RoboDK station: Config_3.rdk

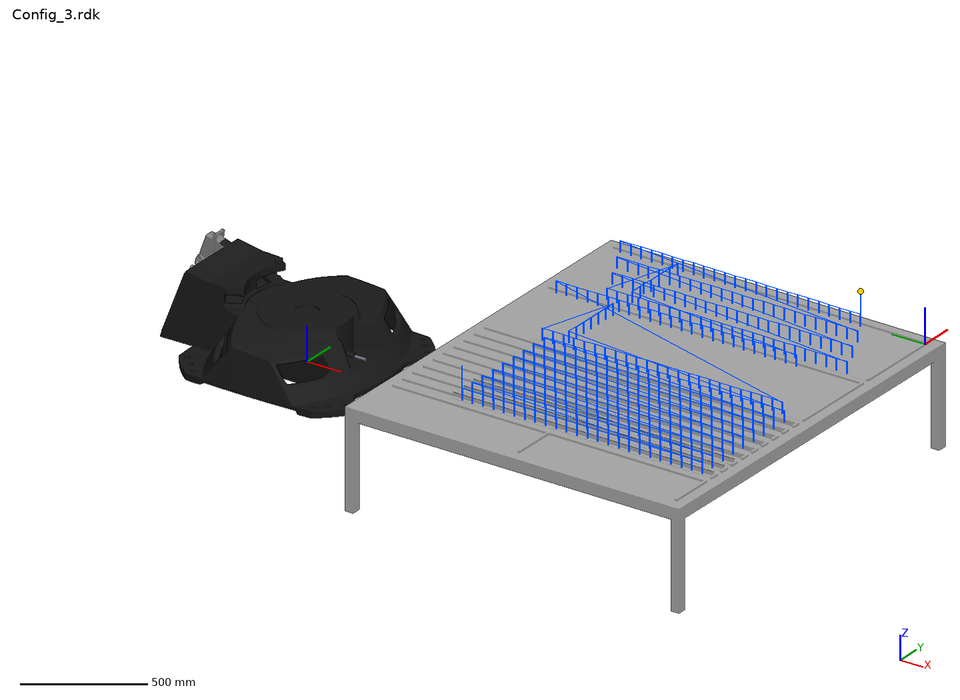
[picture v0: the station drawn from its stored meshes, robots at their saved joint values, targets as dots, program paths as lines]
Station Config_3 (saved by RoboDK 5.2.3). Poses are relative to the parent item; angles as X-Y-Z fixed-axis rotations.
  - frame KUKA KR 210 R2700 extra Base at (0, 0, 0) mm
    - robot KUKA KR 210 R2700 extra: 6 axes, payload 210 kg, reach 2696 mm, repeatability 0.06 mm, weight 1068 kg
        joint limits [-185, -140, -120, -350, -125, -350] to [185, -5, 155, 350, 125, 350]; home [0, -90, 90, 0, 0, 0]; saved at [38.533, -84.893, 130.139, 228.276, 56.581, -211.701]
      - tool Spindle, TCP at (278.6, 0, 88) mm, rotated rx 0 ry 90 rz 0 deg, size 85 x 346.5 x 128 mm
  - frame Corner First Plate at (2495, 660, 510.8) mm, rotated rx 0 ry 0 rz 90 deg
  - object Table 3 at (1700, -800, 455) mm, rotated rx 0 ry 0 rz 90 deg, size 1820 x 1600 x 475 mm, geometry from Table 3.stl
  - object Config_3 at (2495, 660, 510.8) mm, rotated rx 0 ry 0 rz 90 deg
  - machining project Path1 settings: rotZ(0) | rotX(0)*rotY(0) | rotz(0) | onStart | onPathStart | onApproach | onPoint | onRetract | onFinish | SetRPM(%1) | SetTool(%1) | Extruder(%1) | default | default | OutOnMov(%1) | OutOffMov(%1) | onPathFinish | M_RunCode(%1)
  - program Path1 (1131 instructions, listed below)
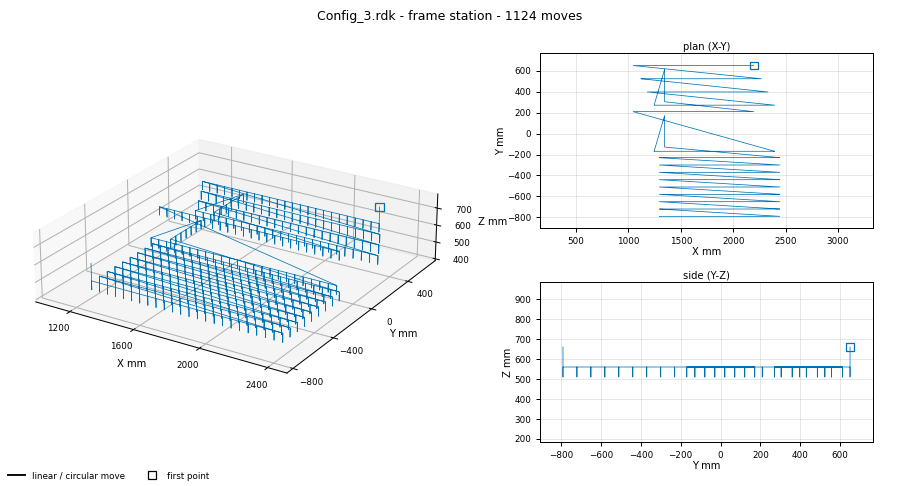
[picture p0: tool path of Config_3.rdk in frame station, 1124 of 1124 moves have a stored position in this frame; points joined in program order, loops and branches not executed]

--- program Path1 (robot KUKA KR 210 R2700 extra) ---
  Smooth(1)
  Set speed (1000.0 mm/s)
  Set Ref.: Corner First Plate
  Set Tool: Spindle
  Show Spindle
  MoveJ 1 to (-10.8, 300, 150) mm, rotated rx 180 ry 0 rz 90 deg; joints [-18.939, -55.022, 87.438, 147.377, 37.015, -152.928]
  MoveL 2 to (-10.8, 300, 150) mm, rotated rx 180 ry 0 rz 90 deg; joints [-18.939, -55.022, 87.438, 147.377, 37.015, -152.928]
  MoveL 3 to (-10.8, 300, 50) mm, rotated rx -180 ry 0 rz 90 deg; joints [-18.939, -52.073, 88.328, 149.877, 40.293, -156.128]
  MoveL 4 to (-10.8, 300, 50) mm, rotated rx -180 ry 0 rz 90 deg; joints [-18.939, -52.073, 88.328, 149.877, 40.293, -156.128]
  Set speed (150.0 mm/s)
  MoveL 5 to (-10.8, 300, -0.5) mm, rotated rx 180 ry 0 rz 90 deg; joints [-18.939, -50.484, 88.62, 150.941, 41.929, -157.54]
  MoveL 6 to (-10.8, 300, 50) mm, rotated rx -180 ry 0 rz 90 deg; joints [-18.939, -52.073, 88.328, 149.877, 40.293, -156.128]
  MoveL 7 to (-10.8, 350, 50) mm, rotated rx 180 ry 0 rz 90 deg; joints [-19.415, -53.906, 91.518, 149.994, 41.659, -156.663]
  MoveL 8 to (-10.8, 350, -0.5) mm, rotated rx 180 ry 0 rz 90 deg; joints [-19.415, -52.267, 91.81, 151.032, 43.339, -158.069]
  MoveL 9 to (-10.8, 350, 50) mm, rotated rx 180 ry 0 rz 90 deg; joints [-19.415, -53.906, 91.518, 149.994, 41.659, -156.663]
  MoveL 10 to (-10.8, 400, 50) mm, rotated rx 180 ry 0 rz 90 deg; joints [-19.914, -55.704, 94.616, 150.026, 42.981, -157.123]
  MoveL 11 to (-10.8, 400, -0.5) mm, rotated rx -180 ry 0 rz 90 deg; joints [-19.914, -54.013, 94.91, 151.042, 44.709, -158.532]
  MoveL 12 to (-10.8, 400, 50) mm, rotated rx 180 ry 0 rz 90 deg; joints [-19.914, -55.704, 94.616, 150.026, 42.981, -157.123]
  MoveL 13 to (-10.8, 450, 50) mm, rotated rx 180 ry 0 rz 90 deg; joints [-20.439, -57.473, 97.631, 149.977, 44.262, -157.517]
  MoveL 14 to (-10.8, 450, -0.5) mm, rotated rx 180 ry 0 rz 90 deg; joints [-20.439, -55.727, 97.926, 150.978, 46.038, -158.936]
  MoveL 15 to (-10.8, 450, 50) mm, rotated rx 180 ry 0 rz 90 deg; joints [-20.439, -57.473, 97.631, 149.977, 44.262, -157.517]
  MoveL 16 to (-10.8, 500, 50) mm, rotated rx -180 ry 0 rz 90 deg; joints [-20.991, -59.217, 100.569, 149.854, 45.504, -157.852]
  MoveL 17 to (-10.8, 500, -0.5) mm, rotated rx 180 ry 0 rz 90 deg; joints [-20.991, -57.414, 100.867, 150.844, 47.331, -159.288]
  MoveL 18 to (-10.8, 500, 50) mm, rotated rx -180 ry 0 rz 90 deg; joints [-20.991, -59.217, 100.569, 149.854, 45.504, -157.852]
  MoveL 19 to (-10.8, 550, 50) mm, rotated rx 180 ry 0 rz 90 deg; joints [-21.572, -60.942, 103.435, 149.66, 46.709, -158.133]
  MoveL 20 to (-10.8, 550, -0.5) mm, rotated rx 180 ry 0 rz 90 deg; joints [-21.572, -59.078, 103.738, 150.643, 48.588, -159.592]
  MoveL 21 to (-10.8, 550, 50) mm, rotated rx 180 ry 0 rz 90 deg; joints [-21.572, -60.942, 103.435, 149.66, 46.709, -158.133]
  MoveL 22 to (-10.8, 600, 50) mm, rotated rx 180 ry 0 rz 90 deg; joints [-22.185, -62.649, 106.236, 149.397, 47.878, -158.362]
  MoveL 23 to (-10.8, 600, -0.5) mm, rotated rx 180 ry 0 rz 90 deg; joints [-22.185, -60.721, 106.543, 150.377, 49.812, -159.851]
  MoveL 24 to (-10.8, 600, 50) mm, rotated rx 180 ry 0 rz 90 deg; joints [-22.185, -62.649, 106.236, 149.397, 47.878, -158.362]
  MoveL 25 to (-10.8, 650, 50) mm, rotated rx 180 ry 0 rz 90 deg; joints [-22.832, -64.344, 108.975, 149.067, 49.013, -158.542]
  MoveL 26 to (-10.8, 650, -0.5) mm, rotated rx 180 ry 0 rz 90 deg; joints [-22.832, -62.348, 109.287, 150.048, 51.003, -160.069]
  MoveL 27 to (-10.8, 650, 50) mm, rotated rx 180 ry 0 rz 90 deg; joints [-22.832, -64.344, 108.975, 149.067, 49.013, -158.542]
  MoveL 28 to (-10.8, 700, 50) mm, rotated rx -180 ry 0 rz 90 deg; joints [-23.515, -66.029, 111.655, 148.669, 50.113, -158.676]
  MoveL 29 to (-10.8, 700, -0.5) mm, rotated rx 180 ry 0 rz 90 deg; joints [-23.515, -63.961, 111.973, 149.655, 52.163, -160.247]
  MoveL 30 to (-10.8, 700, 50) mm, rotated rx -180 ry 0 rz 90 deg; joints [-23.515, -66.029, 111.655, 148.669, 50.113, -158.676]
  MoveL 31 to (-10.8, 750, 50) mm, rotated rx 180 ry 0 rz 90 deg; joints [-24.238, -67.708, 114.279, 148.204, 51.181, -158.763]
  MoveL 32 to (-10.8, 750, -0.5) mm, rotated rx 180 ry 0 rz 90 deg; joints [-24.238, -65.564, 114.604, 149.198, 53.292, -160.386]
  MoveL 33 to (-10.8, 750, 50) mm, rotated rx 180 ry 0 rz 90 deg; joints [-24.238, -67.708, 114.279, 148.204, 51.181, -158.763]
  MoveL 34 to (-10.8, 800, 50) mm, rotated rx -180 ry 0 rz 90 deg; joints [-25.003, -69.384, 116.85, 147.669, 52.216, -158.805]
  MoveL 35 to (-10.8, 800, -0.5) mm, rotated rx 180 ry 0 rz 90 deg; joints [-25.003, -67.159, 117.183, 148.675, 54.391, -160.488]
  MoveL 36 to (-10.8, 800, 50) mm, rotated rx -180 ry 0 rz 90 deg; joints [-25.003, -69.384, 116.85, 147.669, 52.216, -158.805]
  MoveL 37 to (-10.8, 850, 50) mm, rotated rx -180 ry 0 rz 90 deg; joints [-25.816, -71.061, 119.369, 147.064, 53.22, -158.799]
  MoveL 38 to (-10.8, 850, -0.5) mm, rotated rx 180 ry 0 rz 90 deg; joints [-25.816, -68.749, 119.711, 148.085, 55.46, -160.551]
  MoveL 39 to (-10.8, 850, 50) mm, rotated rx -180 ry 0 rz 90 deg; joints [-25.816, -71.061, 119.369, 147.064, 53.22, -158.799]
  MoveL 40 to (-10.8, 900, 50) mm, rotated rx 180 ry 0 rz 90 deg; joints [-26.678, -72.742, 121.838, 146.383, 54.192, -158.746]
  MoveL 41 to (-10.8, 900, -0.5) mm, rotated rx -180 ry 0 rz 90 deg; joints [-26.678, -70.337, 122.19, 147.424, 56.501, -160.575]
  MoveL 42 to (-10.8, 900, 50) mm, rotated rx 180 ry 0 rz 90 deg; joints [-26.678, -72.742, 121.838, 146.383, 54.192, -158.746]
  MoveL 43 to (-10.8, 950, 50) mm, rotated rx -180 ry 0 rz 90 deg; joints [-27.596, -74.43, 124.259, 145.626, 55.132, -158.641]
  MoveL 44 to (-10.8, 950, -0.5) mm, rotated rx -180 ry 0 rz 90 deg; joints [-27.596, -71.926, 124.621, 146.689, 57.513, -160.559]
  MoveL 45 to (-10.8, 950, 50) mm, rotated rx -180 ry 0 rz 90 deg; joints [-27.596, -74.43, 124.259, 145.626, 55.132, -158.641]
  MoveL 46 to (-10.8, 1000, 50) mm, rotated rx 180 ry 0 rz 90 deg; joints [-28.574, -76.128, 126.631, 144.786, 56.043, -158.484]
  MoveL 47 to (-10.8, 1000, -0.5) mm, rotated rx 180 ry 0 rz 90 deg; joints [-28.574, -73.519, 127.005, 145.877, 58.497, -160.501]
  MoveL 48 to (-10.8, 1000, 50) mm, rotated rx 180 ry 0 rz 90 deg; joints [-28.574, -76.128, 126.631, 144.786, 56.043, -158.484]
  MoveL 49 to (-10.8, 1050, 50) mm, rotated rx -180 ry 0 rz 90 deg; joints [-29.617, -77.842, 128.955, 143.858, 56.923, -158.269]
  MoveL 50 to (-10.8, 1050, -0.5) mm, rotated rx 180 ry 0 rz 90 deg; joints [-29.617, -75.119, 129.342, 144.981, 59.453, -160.398]
  MoveL 51 to (-10.8, 1050, 50) mm, rotated rx -180 ry 0 rz 90 deg; joints [-29.617, -77.842, 128.955, 143.858, 56.923, -158.269]
  MoveL 52 to (-10.8, 1100, 50) mm, rotated rx 180 ry 0 rz 90 deg; joints [-30.732, -79.573, 131.231, 142.838, 57.775, -157.992]
  MoveL 53 to (-10.8, 1100, -0.5) mm, rotated rx -180 ry 0 rz 90 deg; joints [-30.732, -76.729, 131.632, 143.997, 60.382, -160.246]
  MoveL 54 to (-10.8, 1100, 50) mm, rotated rx 180 ry 0 rz 90 deg; joints [-30.732, -79.573, 131.231, 142.838, 57.775, -157.992]
  MoveL 55 to (-10.8, 1150, 50) mm, rotated rx 180 ry 0 rz 90 deg; joints [-31.924, -81.327, 133.457, 141.718, 58.599, -157.647]
  MoveL 56 to (-10.8, 1150, -0.5) mm, rotated rx 180 ry 0 rz 90 deg; joints [-31.924, -78.352, 133.874, 142.918, 61.284, -160.042]
  MoveL 57 to (-10.8, 1150, 50) mm, rotated rx 180 ry 0 rz 90 deg; joints [-31.924, -81.327, 133.457, 141.718, 58.599, -157.647]
  MoveL 58 to (-10.8, 1200, 50) mm, rotated rx 180 ry 0 rz 90 deg; joints [-33.202, -83.108, 135.634, 140.49, 59.397, -157.227]
  MoveL 59 to (-10.8, 1200, -0.5) mm, rotated rx 180 ry 0 rz 90 deg; joints [-33.202, -79.993, 136.068, 141.737, 62.161, -159.78]
  MoveL 60 to (-10.8, 1200, 50) mm, rotated rx 180 ry 0 rz 90 deg; joints [-33.202, -83.108, 135.634, 140.49, 59.397, -157.227]
  MoveL 61 to (-10.8, 1250, 50) mm, rotated rx -180 ry 0 rz 90 deg; joints [-34.574, -84.92, 137.758, 139.147, 60.172, -156.726]
  MoveL 62 to (-10.8, 1250, -0.5) mm, rotated rx -180 ry 0 rz 90 deg; joints [-34.574, -81.654, 138.211, 140.446, 63.014, -159.455]
  MoveL 63 to (-10.8, 1250, 50) mm, rotated rx -180 ry 0 rz 90 deg; joints [-34.574, -84.92, 137.758, 139.147, 60.172, -156.726]
  MoveL 64 to (-10.8, 1300, 50) mm, rotated rx 180 ry 0 rz 90 deg; joints [-36.047, -86.767, 139.828, 137.68, 60.929, -156.133]
  MoveL 65 to (-10.8, 1300, -0.5) mm, rotated rx 180 ry 0 rz 90 deg; joints [-36.047, -83.339, 140.302, 139.037, 63.846, -159.059]
  MoveL 66 to (-10.8, 1300, 50) mm, rotated rx 180 ry 0 rz 90 deg; joints [-36.047, -86.767, 139.828, 137.68, 60.929, -156.133]
  MoveL 67 to (-10.8, 1350, 50) mm, rotated rx 180 ry 0 rz 90 deg; joints [-37.633, -88.655, 141.842, 136.078, 61.671, -155.439]
  MoveL 68 to (-10.8, 1350, -0.5) mm, rotated rx 180 ry 0 rz 90 deg; joints [-37.633, -85.052, 142.339, 137.499, 64.659, -158.585]
  MoveL 69 to (-10.8, 1350, 50) mm, rotated rx 180 ry 0 rz 90 deg; joints [-37.633, -88.655, 141.842, 136.078, 61.671, -155.439]
  MoveL 70 to (-10.8, 1400, 50) mm, rotated rx -180 ry 0 rz 90 deg; joints [-39.341, -90.587, 143.795, 134.333, 62.407, -154.634]
  MoveL 71 to (-10.8, 1400, -0.5) mm, rotated rx 180 ry 0 rz 90 deg; joints [-39.341, -86.798, 144.317, 135.822, 65.461, -158.023]
  MoveL 72 to (-10.8, 1400, 50) mm, rotated rx -180 ry 0 rz 90 deg; joints [-39.341, -90.587, 143.795, 134.333, 62.407, -154.634]
  MoveL 73 to (-10.8, 1450, 50) mm, rotated rx 180 ry 0 rz 90 deg; joints [-41.184, -92.567, 145.684, 132.434, 63.147, -153.707]
  MoveL 74 to (-10.8, 1450, -0.5) mm, rotated rx -180 ry 0 rz 90 deg; joints [-41.184, -88.578, 146.233, 133.998, 66.256, -157.364]
  MoveL 75 to (-10.8, 1450, 50) mm, rotated rx 180 ry 0 rz 90 deg; joints [-41.184, -92.567, 145.684, 132.434, 63.147, -153.707]
  MoveL 76 to (-136.94, 226.53, 50) mm, rotated rx -180 ry 0 rz 90 deg; joints [-14.902, -50.749, 86.003, 155.248, 37.896, -160.007]
  MoveL 77 to (-136.94, 226.53, -0.5) mm, rotated rx 180 ry 0 rz 90 deg; joints [-14.902, -49.194, 86.295, 156.194, 39.579, -161.22]
  MoveL 78 to (-136.94, 226.53, 50) mm, rotated rx -180 ry 0 rz 90 deg; joints [-14.902, -50.749, 86.003, 155.248, 37.896, -160.007]
  MoveL 79 to (-136.94, 276.53, 50) mm, rotated rx -180 ry 0 rz 90 deg; joints [-15.273, -52.646, 89.329, 155.434, 39.319, -160.525]
  MoveL 80 to (-136.94, 276.53, -0.5) mm, rotated rx 180 ry 0 rz 90 deg; joints [-15.273, -51.042, 89.62, 156.351, 41.049, -161.724]
  MoveL 81 to (-136.94, 276.53, 50) mm, rotated rx -180 ry 0 rz 90 deg; joints [-15.273, -52.646, 89.329, 155.434, 39.319, -160.525]
  MoveL 82 to (-136.94, 326.53, 50) mm, rotated rx -180 ry 0 rz 90 deg; joints [-15.663, -54.506, 92.556, 155.538, 40.691, -160.969]
  MoveL 83 to (-136.94, 326.53, -0.5) mm, rotated rx -180 ry 0 rz 90 deg; joints [-15.663, -52.85, 92.848, 156.432, 42.471, -162.163]
  MoveL 84 to (-136.94, 326.53, 50) mm, rotated rx -180 ry 0 rz 90 deg; joints [-15.663, -54.506, 92.556, 155.538, 40.691, -160.969]
  MoveL 85 to (-136.94, 376.53, 50) mm, rotated rx 180 ry 0 rz 90 deg; joints [-16.072, -56.334, 95.694, 155.568, 42.016, -161.349]
  MoveL 86 to (-136.94, 376.53, -0.5) mm, rotated rx -180 ry 0 rz 90 deg; joints [-16.072, -54.624, 95.988, 156.444, 43.847, -162.545]
  MoveL 87 to (-136.94, 376.53, 50) mm, rotated rx 180 ry 0 rz 90 deg; joints [-16.072, -56.334, 95.694, 155.568, 42.016, -161.349]
  MoveL 88 to (-136.94, 426.53, 50) mm, rotated rx 180 ry 0 rz 90 deg; joints [-16.503, -58.136, 98.751, 155.529, 43.296, -161.673]
  MoveL 89 to (-136.94, 426.53, -0.5) mm, rotated rx -180 ry 0 rz 90 deg; joints [-16.503, -56.369, 99.048, 156.392, 45.18, -162.878]
  MoveL 90 to (-136.94, 426.53, 50) mm, rotated rx 180 ry 0 rz 90 deg; joints [-16.503, -58.136, 98.751, 155.529, 43.296, -161.673]
  MoveL 91 to (-136.94, 476.53, 50) mm, rotated rx 180 ry 0 rz 90 deg; joints [-16.957, -59.916, 101.734, 155.426, 44.532, -161.945]
  MoveL 92 to (-136.94, 476.53, -0.5) mm, rotated rx -180 ry 0 rz 90 deg; joints [-16.957, -58.088, 102.034, 156.281, 46.473, -163.165]
  MoveL 93 to (-136.94, 476.53, 50) mm, rotated rx 180 ry 0 rz 90 deg; joints [-16.957, -59.916, 101.734, 155.426, 44.532, -161.945]
  MoveL 94 to (-136.94, 526.53, 50) mm, rotated rx 180 ry 0 rz 90 deg; joints [-17.435, -61.679, 104.649, 155.262, 45.726, -162.17]
  MoveL 95 to (-136.94, 526.53, -0.5) mm, rotated rx 180 ry 0 rz 90 deg; joints [-17.435, -59.788, 104.954, 156.113, 47.727, -163.411]
  MoveL 96 to (-136.94, 526.53, 50) mm, rotated rx 180 ry 0 rz 90 deg; joints [-17.435, -61.679, 104.649, 155.262, 45.726, -162.17]
  MoveL 97 to (-136.94, 576.53, 50) mm, rotated rx -180 ry 0 rz 90 deg; joints [-17.941, -63.429, 107.501, 155.038, 46.88, -162.35]
  MoveL 98 to (-136.94, 576.53, -0.5) mm, rotated rx -180 ry 0 rz 90 deg; joints [-17.941, -61.47, 107.811, 155.889, 48.944, -163.619]
  MoveL 99 to (-136.94, 576.53, 50) mm, rotated rx -180 ry 0 rz 90 deg; joints [-17.941, -63.429, 107.501, 155.038, 46.88, -162.35]
  MoveL 100 to (-136.94, 626.53, 50) mm, rotated rx -180 ry 0 rz 90 deg; joints [-18.476, -65.17, 110.295, 154.756, 47.994, -162.488]
  MoveL 101 to (-136.94, 626.53, -0.5) mm, rotated rx -180 ry 0 rz 90 deg; joints [-18.476, -63.14, 110.61, 155.61, 50.124, -163.791]
  MoveL 102 to (-136.94, 626.53, 50) mm, rotated rx -180 ry 0 rz 90 deg; joints [-18.476, -65.17, 110.295, 154.756, 47.994, -162.488]
  MoveL 103 to (-136.94, 676.53, 50) mm, rotated rx -180 ry 0 rz 90 deg; joints [-19.042, -66.907, 113.033, 154.415, 49.069, -162.584]
  MoveL 104 to (-136.94, 676.53, -0.5) mm, rotated rx 180 ry 0 rz 90 deg; joints [-19.042, -64.8, 113.355, 155.276, 51.268, -163.929]
  MoveL 105 to (-136.94, 676.53, 50) mm, rotated rx -180 ry 0 rz 90 deg; joints [-19.042, -66.907, 113.033, 154.415, 49.069, -162.584]
  MoveL 106 to (-136.94, 726.53, 50) mm, rotated rx 180 ry 0 rz 90 deg; joints [-19.643, -68.643, 115.719, 154.014, 50.104, -162.639]
  MoveL 107 to (-136.94, 726.53, -0.5) mm, rotated rx -180 ry 0 rz 90 deg; joints [-19.643, -66.454, 116.049, 154.886, 52.376, -164.032]
  MoveL 108 to (-136.94, 726.53, 50) mm, rotated rx 180 ry 0 rz 90 deg; joints [-19.643, -68.643, 115.719, 154.014, 50.104, -162.639]
  MoveL 109 to (-136.94, 776.53, 50) mm, rotated rx 180 ry 0 rz 90 deg; joints [-20.281, -70.382, 118.355, 153.551, 51.099, -162.652]
  MoveL 110 to (-136.94, 776.53, -0.5) mm, rotated rx -180 ry 0 rz 90 deg; joints [-20.281, -68.106, 118.694, 154.439, 53.45, -164.101]
  MoveL 111 to (-136.94, 776.53, 50) mm, rotated rx 180 ry 0 rz 90 deg; joints [-20.281, -70.382, 118.355, 153.551, 51.099, -162.652]
  MoveL 112 to (-136.94, 826.53, 50) mm, rotated rx 180 ry 0 rz 90 deg; joints [-20.96, -72.129, 120.945, 153.024, 52.055, -162.621]
  MoveL 113 to (-136.94, 826.53, -0.5) mm, rotated rx 180 ry 0 rz 90 deg; joints [-20.96, -69.759, 121.293, 153.93, 54.487, -164.135]
  MoveL 114 to (-136.94, 826.53, 50) mm, rotated rx 180 ry 0 rz 90 deg; joints [-20.96, -72.129, 120.945, 153.024, 52.055, -162.621]
  MoveL 115 to (-136.94, 876.53, 50) mm, rotated rx -180 ry 0 rz 90 deg; joints [-21.684, -73.888, 123.489, 152.43, 52.969, -162.544]
  MoveL 116 to (-136.94, 876.53, -0.5) mm, rotated rx -180 ry 0 rz 90 deg; joints [-21.684, -71.417, 123.848, 153.359, 55.489, -164.134]
  MoveL 117 to (-136.94, 876.53, 50) mm, rotated rx -180 ry 0 rz 90 deg; joints [-21.684, -73.888, 123.489, 152.43, 52.969, -162.544]
  MoveL 118 to (-136.94, 926.53, 50) mm, rotated rx -180 ry 0 rz 90 deg; joints [-22.457, -75.664, 125.989, 151.763, 53.842, -162.419]
  MoveL 119 to (-136.94, 926.53, -0.5) mm, rotated rx 180 ry 0 rz 90 deg; joints [-22.457, -73.084, 126.36, 152.721, 56.453, -164.094]
  MoveL 120 to (-136.94, 926.53, 50) mm, rotated rx -180 ry 0 rz 90 deg; joints [-22.457, -75.664, 125.989, 151.763, 53.842, -162.419]
  MoveL 121 to (-136.94, 976.53, 50) mm, rotated rx -180 ry 0 rz 90 deg; joints [-23.284, -77.462, 128.446, 151.02, 54.671, -162.241]
  MoveL 122 to (-136.94, 976.53, -0.5) mm, rotated rx 180 ry 0 rz 90 deg; joints [-23.284, -74.765, 128.83, 152.01, 57.38, -164.013]
  MoveL 123 to (-136.94, 976.53, 50) mm, rotated rx -180 ry 0 rz 90 deg; joints [-23.284, -77.462, 128.446, 151.02, 54.671, -162.241]
  MoveL 124 to (-136.94, 1026.53, 50) mm, rotated rx 180 ry 0 rz 90 deg; joints [-24.17, -79.288, 130.861, 150.192, 55.456, -162.004]
  MoveL 125 to (-136.94, 1026.53, -0.5) mm, rotated rx -180 ry 0 rz 90 deg; joints [-24.17, -76.464, 131.259, 151.222, 58.267, -163.887]
  MoveL 126 to (-136.94, 1026.53, 50) mm, rotated rx 180 ry 0 rz 90 deg; joints [-24.17, -79.288, 130.861, 150.192, 55.456, -162.004]
  MoveL 127 to (-136.94, 1076.53, 50) mm, rotated rx -180 ry 0 rz 90 deg; joints [-25.123, -81.148, 133.233, 149.274, 56.195, -161.702]
  MoveL 128 to (-136.94, 1076.53, -0.5) mm, rotated rx 180 ry 0 rz 90 deg; joints [-25.123, -78.186, 133.648, 150.349, 59.114, -163.711]
  MoveL 129 to (-136.94, 1076.53, 50) mm, rotated rx -180 ry 0 rz 90 deg; joints [-25.123, -81.148, 133.233, 149.274, 56.195, -161.702]
  MoveL 130 to (-136.94, 1126.53, 50) mm, rotated rx 180 ry 0 rz 90 deg; joints [-26.147, -83.049, 135.562, 148.256, 56.887, -161.326]
  MoveL 131 to (-136.94, 1126.53, -0.5) mm, rotated rx 180 ry 0 rz 90 deg; joints [-26.147, -79.938, 135.996, 149.385, 59.919, -163.48]
  MoveL 132 to (-136.94, 1126.53, 50) mm, rotated rx 180 ry 0 rz 90 deg; joints [-26.147, -83.049, 135.562, 148.256, 56.887, -161.326]
  MoveL 133 to (-136.94, 1176.53, 50) mm, rotated rx 180 ry 0 rz 90 deg; joints [-27.253, -84.999, 137.848, 147.128, 57.529, -160.866]
  MoveL 134 to (-136.94, 1176.53, -0.5) mm, rotated rx -180 ry 0 rz 90 deg; joints [-27.253, -81.726, 138.302, 148.319, 60.68, -163.185]
  MoveL 135 to (-136.94, 1176.53, 50) mm, rotated rx 180 ry 0 rz 90 deg; joints [-27.253, -84.999, 137.848, 147.128, 57.529, -160.866]
  MoveL 136 to (-136.94, 1226.53, 50) mm, rotated rx -180 ry 0 rz 90 deg; joints [-28.447, -87.007, 140.09, 145.877, 58.121, -160.309]
  MoveL 137 to (-136.94, 1226.53, -0.5) mm, rotated rx 180 ry 0 rz 90 deg; joints [-28.447, -83.557, 140.567, 147.141, 61.396, -162.817]
  MoveL 138 to (-136.94, 1226.53, 50) mm, rotated rx -180 ry 0 rz 90 deg; joints [-28.447, -87.007, 140.09, 145.877, 58.121, -160.309]
  MoveL 139 to (-136.94, 1276.53, 50) mm, rotated rx -180 ry 0 rz 90 deg; joints [-29.742, -89.084, 142.285, 144.491, 58.661, -159.64]
  MoveL 140 to (-136.94, 1276.53, -0.5) mm, rotated rx -180 ry 0 rz 90 deg; joints [-29.742, -85.441, 142.787, 145.839, 62.064, -162.364]
  MoveL 141 to (-136.94, 1276.53, 50) mm, rotated rx -180 ry 0 rz 90 deg; joints [-29.742, -89.084, 142.285, 144.491, 58.661, -159.64]
  MoveL 142 to (-136.94, 1326.53, 50) mm, rotated rx -180 ry 0 rz 90 deg; joints [-31.147, -91.241, 144.432, 142.952, 59.151, -158.84]
  MoveL 143 to (-136.94, 1326.53, -0.5) mm, rotated rx -180 ry 0 rz 90 deg; joints [-31.147, -87.387, 144.962, 144.398, 62.685, -161.812]
  MoveL 144 to (-136.94, 1326.53, 50) mm, rotated rx -180 ry 0 rz 90 deg; joints [-31.147, -91.241, 144.432, 142.952, 59.151, -158.84]
  MoveL 145 to (-136.94, 1376.53, 50) mm, rotated rx -180 ry 0 rz 90 deg; joints [-32.677, -93.491, 146.526, 141.244, 59.593, -157.887]
  MoveL 146 to (-136.94, 1376.53, -0.5) mm, rotated rx 180 ry 0 rz 90 deg; joints [-32.677, -89.406, 147.089, 142.802, 63.257, -161.143]
  MoveL 147 to (-136.94, 1376.53, 50) mm, rotated rx -180 ry 0 rz 90 deg; joints [-32.677, -93.491, 146.526, 141.244, 59.593, -157.887]
  MoveL 148 to (-263.08, 163.47, 50) mm, rotated rx 180 ry 0 rz 90 deg; joints [-11.071, -49.424, 83.663, 160.824, 35.776, -164.244]
  MoveL 149 to (-263.08, 163.47, -0.5) mm, rotated rx 180 ry 0 rz 90 deg; joints [-11.071, -47.902, 83.955, 161.61, 37.493, -165.223]
  MoveL 150 to (-263.08, 163.47, 50) mm, rotated rx 180 ry 0 rz 90 deg; joints [-11.071, -49.424, 83.663, 160.824, 35.776, -164.244]
  MoveL 151 to (-263.08, 213.47, 50) mm, rotated rx -180 ry 0 rz 90 deg; joints [-11.344, -51.379, 87.111, 161.042, 37.26, -164.709]
  MoveL 152 to (-263.08, 213.47, -0.5) mm, rotated rx 180 ry 0 rz 90 deg; joints [-11.344, -49.808, 87.403, 161.797, 39.025, -165.67]
  MoveL 153 to (-263.08, 213.47, 50) mm, rotated rx -180 ry 0 rz 90 deg; joints [-11.344, -51.379, 87.111, 161.042, 37.26, -164.709]
  MoveL 154 to (-263.08, 263.47, 50) mm, rotated rx -180 ry 0 rz 90 deg; joints [-11.63, -53.292, 90.454, 161.185, 38.687, -165.107]
  MoveL 155 to (-263.08, 263.47, -0.5) mm, rotated rx 180 ry 0 rz 90 deg; joints [-11.63, -51.671, 90.745, 161.917, 40.502, -166.057]
  MoveL 156 to (-263.08, 263.47, 50) mm, rotated rx -180 ry 0 rz 90 deg; joints [-11.63, -53.292, 90.454, 161.185, 38.687, -165.107]
  MoveL 157 to (-263.08, 313.47, 50) mm, rotated rx -180 ry 0 rz 90 deg; joints [-11.931, -55.17, 93.701, 161.263, 40.059, -165.446]
  MoveL 158 to (-263.08, 313.47, -0.5) mm, rotated rx -180 ry 0 rz 90 deg; joints [-11.931, -53.496, 93.994, 161.977, 41.927, -166.392]
  MoveL 159 to (-263.08, 313.47, 50) mm, rotated rx -180 ry 0 rz 90 deg; joints [-11.931, -55.17, 93.701, 161.263, 40.059, -165.446]
  MoveL 160 to (-263.08, 363.47, 50) mm, rotated rx 180 ry 0 rz 90 deg; joints [-12.247, -57.02, 96.862, 161.283, 41.38, -165.736]
  MoveL 161 to (-263.08, 363.47, -0.5) mm, rotated rx -180 ry 0 rz 90 deg; joints [-12.247, -55.289, 97.157, 161.983, 43.303, -166.684]
  MoveL 162 to (-263.08, 363.47, 50) mm, rotated rx 180 ry 0 rz 90 deg; joints [-12.247, -57.02, 96.862, 161.283, 41.38, -165.736]
  MoveL 163 to (-263.08, 413.47, 50) mm, rotated rx -180 ry 0 rz 90 deg; joints [-12.581, -58.845, 99.945, 161.248, 42.653, -165.981]
  MoveL 164 to (-263.08, 413.47, -0.5) mm, rotated rx 180 ry 0 rz 90 deg; joints [-12.581, -57.055, 100.243, 161.94, 44.634, -166.936]
  MoveL 165 to (-263.08, 413.47, 50) mm, rotated rx -180 ry 0 rz 90 deg; joints [-12.581, -58.845, 99.945, 161.248, 42.653, -165.981]
  MoveL 166 to (-263.08, 463.47, 50) mm, rotated rx 180 ry 0 rz 90 deg; joints [-12.933, -60.652, 102.957, 161.162, 43.878, -166.184]
  MoveL 167 to (-263.08, 463.47, -0.5) mm, rotated rx 180 ry 0 rz 90 deg; joints [-12.933, -58.799, 103.259, 161.848, 45.922, -167.153]
  MoveL 168 to (-263.08, 463.47, 50) mm, rotated rx 180 ry 0 rz 90 deg; joints [-12.933, -60.652, 102.957, 161.162, 43.878, -166.184]
  MoveL 169 to (-263.08, 513.47, 50) mm, rotated rx -180 ry 0 rz 90 deg; joints [-13.304, -62.446, 105.904, 161.028, 45.058, -166.35]
  MoveL 170 to (-263.08, 513.47, -0.5) mm, rotated rx -180 ry 0 rz 90 deg; joints [-13.304, -60.526, 106.211, 161.712, 47.168, -167.337]
  MoveL 171 to (-263.08, 513.47, 50) mm, rotated rx -180 ry 0 rz 90 deg; joints [-13.304, -62.446, 105.904, 161.028, 45.058, -166.35]
  MoveL 172 to (-263.08, 563.47, 50) mm, rotated rx 180 ry 0 rz 90 deg; joints [-13.698, -64.23, 108.792, 160.845, 46.193, -166.48]
  MoveL 173 to (-263.08, 563.47, -0.5) mm, rotated rx 180 ry 0 rz 90 deg; joints [-13.698, -62.238, 109.104, 161.531, 48.373, -167.491]
  MoveL 174 to (-263.08, 563.47, 50) mm, rotated rx 180 ry 0 rz 90 deg; joints [-13.698, -64.23, 108.792, 160.845, 46.193, -166.48]
  MoveL 175 to (-263.08, 613.47, 50) mm, rotated rx 180 ry 0 rz 90 deg; joints [-14.114, -66.009, 111.623, 160.615, 47.283, -166.575]
  MoveL 176 to (-263.08, 613.47, -0.5) mm, rotated rx -180 ry 0 rz 90 deg; joints [-14.114, -63.942, 111.942, 161.306, 49.539, -167.616]
  MoveL 177 to (-263.08, 613.47, 50) mm, rotated rx 180 ry 0 rz 90 deg; joints [-14.114, -66.009, 111.623, 160.615, 47.283, -166.575]
  MoveL 178 to (-263.08, 663.47, 50) mm, rotated rx 180 ry 0 rz 90 deg; joints [-14.557, -67.788, 114.403, 160.338, 48.329, -166.637]
  MoveL 179 to (-263.08, 663.47, -0.5) mm, rotated rx 180 ry 0 rz 90 deg; joints [-14.557, -65.64, 114.729, 161.037, 50.664, -167.713]
  MoveL 180 to (-263.08, 663.47, 50) mm, rotated rx 180 ry 0 rz 90 deg; joints [-14.557, -67.788, 114.403, 160.338, 48.329, -166.637]
  MoveL 181 to (-263.08, 713.47, 50) mm, rotated rx -180 ry 0 rz 90 deg; joints [-15.027, -69.572, 117.134, 160.011, 49.329, -166.663]
  MoveL 182 to (-263.08, 713.47, -0.5) mm, rotated rx 180 ry 0 rz 90 deg; joints [-15.027, -67.337, 117.468, 160.722, 51.749, -167.781]
  MoveL 183 to (-263.08, 713.47, 50) mm, rotated rx -180 ry 0 rz 90 deg; joints [-15.027, -69.572, 117.134, 160.011, 49.329, -166.663]
  MoveL 184 to (-263.08, 763.47, 50) mm, rotated rx 180 ry 0 rz 90 deg; joints [-15.528, -71.365, 119.819, 159.633, 50.282, -166.654]
  MoveL 185 to (-263.08, 763.47, -0.5) mm, rotated rx -180 ry 0 rz 90 deg; joints [-15.528, -69.036, 120.163, 160.359, 52.793, -167.822]
  MoveL 186 to (-263.08, 763.47, 50) mm, rotated rx 180 ry 0 rz 90 deg; joints [-15.528, -71.365, 119.819, 159.633, 50.282, -166.654]
  MoveL 187 to (-263.08, 813.47, 50) mm, rotated rx -180 ry 0 rz 90 deg; joints [-16.063, -73.172, 122.461, 159.201, 51.187, -166.608]
  MoveL 188 to (-263.08, 813.47, -0.5) mm, rotated rx 180 ry 0 rz 90 deg; joints [-16.063, -70.743, 122.815, 159.947, 53.796, -167.833]
  MoveL 189 to (-263.08, 813.47, 50) mm, rotated rx -180 ry 0 rz 90 deg; joints [-16.063, -73.172, 122.461, 159.201, 51.187, -166.608]
  MoveL 190 to (-263.08, 863.47, 50) mm, rotated rx 180 ry 0 rz 90 deg; joints [-16.634, -75, 125.062, 158.711, 52.042, -166.522]
  MoveL 191 to (-263.08, 863.47, -0.5) mm, rotated rx 180 ry 0 rz 90 deg; joints [-16.634, -72.461, 125.428, 159.481, 54.755, -167.813]
  MoveL 192 to (-263.08, 863.47, 50) mm, rotated rx 180 ry 0 rz 90 deg; joints [-16.634, -75, 125.062, 158.711, 52.042, -166.522]
  MoveL 193 to (-263.08, 913.47, 50) mm, rotated rx -180 ry 0 rz 90 deg; joints [-17.247, -76.854, 127.623, 158.16, 52.843, -166.392]
  MoveL 194 to (-263.08, 913.47, -0.5) mm, rotated rx -180 ry 0 rz 90 deg; joints [-17.247, -74.197, 128.003, 158.959, 55.669, -167.759]
  MoveL 195 to (-263.08, 913.47, 50) mm, rotated rx -180 ry 0 rz 90 deg; joints [-17.247, -76.854, 127.623, 158.16, 52.843, -166.392]
  MoveL 196 to (-263.08, 963.47, 50) mm, rotated rx -180 ry 0 rz 90 deg; joints [-17.905, -78.741, 130.146, 157.541, 53.587, -166.213]
  MoveL 197 to (-263.08, 963.47, -0.5) mm, rotated rx -180 ry 0 rz 90 deg; joints [-17.905, -75.956, 130.54, 158.375, 56.534, -167.669]
  MoveL 198 to (-263.08, 963.47, 50) mm, rotated rx -180 ry 0 rz 90 deg; joints [-17.905, -78.741, 130.146, 157.541, 53.587, -166.213]
  MoveL 199 to (-263.08, 1013.47, 50) mm, rotated rx -180 ry 0 rz 90 deg; joints [-18.613, -80.67, 132.632, 156.848, 54.271, -165.979]
  MoveL 200 to (-263.08, 1013.47, -0.5) mm, rotated rx -180 ry 0 rz 90 deg; joints [-18.613, -77.744, 133.043, 157.723, 57.348, -167.537]
  MoveL 201 to (-263.08, 1013.47, 50) mm, rotated rx -180 ry 0 rz 90 deg; joints [-18.613, -80.67, 132.632, 156.848, 54.271, -165.979]
  MoveL 202 to (-263.08, 1063.47, 50) mm, rotated rx 180 ry 0 rz 90 deg; joints [-19.377, -82.649, 135.08, 156.072, 54.888, -165.682]
  MoveL 203 to (-263.08, 1063.47, -0.5) mm, rotated rx -180 ry 0 rz 90 deg; joints [-19.377, -79.57, 135.51, 156.997, 58.107, -167.358]
  MoveL 204 to (-263.08, 1063.47, 50) mm, rotated rx 180 ry 0 rz 90 deg; joints [-19.377, -82.649, 135.08, 156.072, 54.888, -165.682]
  MoveL 205 to (-263.08, 1113.47, 50) mm, rotated rx 180 ry 0 rz 90 deg; joints [-20.205, -84.689, 137.492, 155.203, 55.434, -165.312]
  MoveL 206 to (-263.08, 1113.47, -0.5) mm, rotated rx -180 ry 0 rz 90 deg; joints [-20.205, -81.443, 137.943, 156.187, 58.804, -167.124]
  MoveL 207 to (-263.08, 1113.47, 50) mm, rotated rx 180 ry 0 rz 90 deg; joints [-20.205, -84.689, 137.492, 155.203, 55.434, -165.312]
  MoveL 208 to (-263.08, 1163.47, 50) mm, rotated rx 180 ry 0 rz 90 deg; joints [-21.102, -86.803, 139.868, 154.229, 55.901, -164.855]
  MoveL 209 to (-263.08, 1163.47, -0.5) mm, rotated rx -180 ry 0 rz 90 deg; joints [-21.102, -83.372, 140.342, 155.283, 59.435, -166.826]
  MoveL 210 to (-263.08, 1163.47, 50) mm, rotated rx 180 ry 0 rz 90 deg; joints [-21.102, -86.803, 139.868, 154.229, 55.901, -164.855]
  MoveL 211 to (-263.08, 1213.47, 50) mm, rotated rx -180 ry 0 rz 90 deg; joints [-22.079, -89.006, 142.205, 153.134, 56.282, -164.294]
  MoveL 212 to (-263.08, 1213.47, -0.5) mm, rotated rx -180 ry 0 rz 90 deg; joints [-22.079, -85.37, 142.706, 154.274, 59.991, -166.451]
  MoveL 213 to (-263.08, 1213.47, 50) mm, rotated rx -180 ry 0 rz 90 deg; joints [-22.079, -89.006, 142.205, 153.134, 56.282, -164.294]
  MoveL 214 to (-263.08, 1263.47, 50) mm, rotated rx -180 ry 0 rz 90 deg; joints [-23.145, -91.315, 144.503, 151.901, 56.567, -163.607]
  MoveL 215 to (-263.08, 1263.47, -0.5) mm, rotated rx -180 ry 0 rz 90 deg; joints [-23.145, -87.453, 145.035, 153.143, 60.465, -165.984]
  MoveL 216 to (-263.08, 1263.47, 50) mm, rotated rx -180 ry 0 rz 90 deg; joints [-23.145, -91.315, 144.503, 151.901, 56.567, -163.607]
  MoveL 217 to (-263.08, 1313.47, 50) mm, rotated rx 180 ry 0 rz 90 deg; joints [-24.313, -93.752, 146.76, 150.505, 56.747, -162.768]
  MoveL 218 to (-263.08, 1313.47, -0.5) mm, rotated rx -180 ry 0 rz 90 deg; joints [-24.313, -89.64, 147.327, 151.871, 60.847, -165.403]
  MoveL 219 to (-263.08, 1313.47, 50) mm, rotated rx 180 ry 0 rz 90 deg; joints [-24.313, -93.752, 146.76, 150.505, 56.747, -162.768]
  MoveL 220 to (-389.22, 100, 50) mm, rotated rx 180 ry 0 rz 90 deg; joints [-7.375, -47.693, 80.584, 166.594, 33.617, -168.773]
  MoveL 221 to (-389.22, 100, -0.5) mm, rotated rx 180 ry 0 rz 90 deg; joints [-7.375, -46.211, 80.878, 167.18, 35.346, -169.485]
  MoveL 222 to (-389.22, 100, 50) mm, rotated rx 180 ry 0 rz 90 deg; joints [-7.375, -47.693, 80.584, 166.594, 33.617, -168.773]
  MoveL 223 to (-389.22, 150, 50) mm, rotated rx -180 ry 0 rz 90 deg; joints [-7.554, -49.71, 84.17, 166.81, 35.178, -169.156]
  MoveL 224 to (-389.22, 150, -0.5) mm, rotated rx -180 ry 0 rz 90 deg; joints [-7.554, -48.181, 84.463, 167.369, 36.953, -169.847]
  MoveL 225 to (-389.22, 150, 50) mm, rotated rx -180 ry 0 rz 90 deg; joints [-7.554, -49.71, 84.17, 166.81, 35.178, -169.156]
  MoveL 226 to (-389.22, 200, 50) mm, rotated rx 180 ry 0 rz 90 deg; joints [-7.741, -51.679, 87.638, 166.966, 36.673, -169.482]
  MoveL 227 to (-389.22, 200, -0.5) mm, rotated rx -180 ry 0 rz 90 deg; joints [-7.741, -50.101, 87.93, 167.503, 38.496, -170.159]
  MoveL 228 to (-389.22, 200, 50) mm, rotated rx 180 ry 0 rz 90 deg; joints [-7.741, -51.679, 87.638, 166.966, 36.673, -169.482]
  MoveL 229 to (-389.22, 250, 50) mm, rotated rx 180 ry 0 rz 90 deg; joints [-7.938, -53.608, 91.001, 167.069, 38.106, -169.759]
  MoveL 230 to (-389.22, 250, -0.5) mm, rotated rx -180 ry 0 rz 90 deg; joints [-7.938, -51.977, 91.293, 167.589, 39.981, -170.428]
  MoveL 231 to (-389.22, 250, 50) mm, rotated rx 180 ry 0 rz 90 deg; joints [-7.938, -53.608, 91.001, 167.069, 38.106, -169.759]
  MoveL 232 to (-389.22, 300, 50) mm, rotated rx -180 ry 0 rz 90 deg; joints [-8.145, -55.502, 94.271, 167.126, 39.482, -169.995]
  MoveL 233 to (-389.22, 300, -0.5) mm, rotated rx 180 ry 0 rz 90 deg; joints [-8.145, -53.818, 94.564, 167.633, 41.413, -170.662]
  MoveL 234 to (-389.22, 300, 50) mm, rotated rx -180 ry 0 rz 90 deg; joints [-8.145, -55.502, 94.271, 167.126, 39.482, -169.995]
  MoveL 235 to (-389.22, 350, 50) mm, rotated rx -180 ry 0 rz 90 deg; joints [-8.363, -57.37, 97.455, 167.14, 40.804, -170.196]
  MoveL 236 to (-389.22, 350, -0.5) mm, rotated rx 180 ry 0 rz 90 deg; joints [-8.363, -55.627, 97.751, 167.638, 42.793, -170.863]
  MoveL 237 to (-389.22, 350, 50) mm, rotated rx -180 ry 0 rz 90 deg; joints [-8.363, -57.37, 97.455, 167.14, 40.804, -170.196]
  MoveL 238 to (-389.22, 400, 50) mm, rotated rx 180 ry 0 rz 90 deg; joints [-8.593, -59.215, 100.564, 167.117, 42.075, -170.365]
  MoveL 239 to (-389.22, 400, -0.5) mm, rotated rx -180 ry 0 rz 90 deg; joints [-8.593, -57.412, 100.863, 167.608, 44.126, -171.038]
  MoveL 240 to (-389.22, 400, 50) mm, rotated rx 180 ry 0 rz 90 deg; joints [-8.593, -59.215, 100.564, 167.117, 42.075, -170.365]
  MoveL 241 to (-389.22, 450, 50) mm, rotated rx -180 ry 0 rz 90 deg; joints [-8.835, -61.043, 103.604, 167.057, 43.295, -170.504]
  MoveL 242 to (-389.22, 450, -0.5) mm, rotated rx 180 ry 0 rz 90 deg; joints [-8.835, -59.176, 103.906, 167.545, 45.413, -171.187]
  MoveL 243 to (-389.22, 450, 50) mm, rotated rx -180 ry 0 rz 90 deg; joints [-8.835, -61.043, 103.604, 167.057, 43.295, -170.504]
  MoveL 244 to (-389.22, 500, 50) mm, rotated rx -180 ry 0 rz 90 deg; joints [-9.092, -62.86, 106.58, 166.962, 44.467, -170.617]
  MoveL 245 to (-389.22, 500, -0.5) mm, rotated rx 180 ry 0 rz 90 deg; joints [-9.092, -60.924, 106.887, 167.45, 46.655, -171.312]
  MoveL 246 to (-389.22, 500, 50) mm, rotated rx -180 ry 0 rz 90 deg; joints [-9.092, -62.86, 106.58, 166.962, 44.467, -170.617]
  MoveL 247 to (-389.22, 550, 50) mm, rotated rx -180 ry 0 rz 90 deg; joints [-9.364, -64.671, 109.498, 166.834, 45.59, -170.703]
  MoveL 248 to (-389.22, 550, -0.5) mm, rotated rx 180 ry 0 rz 90 deg; joints [-9.364, -62.661, 109.811, 167.323, 47.855, -171.417]
  MoveL 249 to (-389.22, 550, 50) mm, rotated rx -180 ry 0 rz 90 deg; joints [-9.364, -64.671, 109.498, 166.834, 45.59, -170.703]
  MoveL 250 to (-389.22, 600, 50) mm, rotated rx -180 ry 0 rz 90 deg; joints [-9.653, -66.479, 112.362, 166.671, 46.665, -170.765]
  MoveL 251 to (-389.22, 600, -0.5) mm, rotated rx -180 ry 0 rz 90 deg; joints [-9.653, -64.391, 112.682, 167.165, 49.011, -171.501]
  MoveL 252 to (-389.22, 600, 50) mm, rotated rx -180 ry 0 rz 90 deg; joints [-9.653, -66.479, 112.362, 166.671, 46.665, -170.765]
  MoveL 253 to (-389.22, 650, 50) mm, rotated rx -180 ry 0 rz 90 deg; joints [-9.96, -68.29, 115.177, 166.474, 47.69, -170.802]
  MoveL 254 to (-389.22, 650, -0.5) mm, rotated rx 180 ry 0 rz 90 deg; joints [-9.96, -66.118, 115.505, 166.975, 50.123, -171.564]
  MoveL 255 to (-389.22, 650, 50) mm, rotated rx -180 ry 0 rz 90 deg; joints [-9.96, -68.29, 115.177, 166.474, 47.69, -170.802]
  MoveL 256 to (-389.22, 700, 50) mm, rotated rx 180 ry 0 rz 90 deg; joints [-10.287, -70.109, 117.946, 166.242, 48.665, -170.814]
  MoveL 257 to (-389.22, 700, -0.5) mm, rotated rx 180 ry 0 rz 90 deg; joints [-10.287, -67.847, 118.282, 166.753, 51.192, -171.607]
  MoveL 258 to (-389.22, 700, 50) mm, rotated rx 180 ry 0 rz 90 deg; joints [-10.287, -70.109, 117.946, 166.242, 48.665, -170.814]
  MoveL 259 to (-389.22, 750, 50) mm, rotated rx 180 ry 0 rz 90 deg; joints [-10.635, -71.942, 120.671, 165.972, 49.587, -170.8]
  MoveL 260 to (-389.22, 750, -0.5) mm, rotated rx -180 ry 0 rz 90 deg; joints [-10.635, -69.582, 121.018, 166.496, 52.216, -171.63]
  MoveL 261 to (-389.22, 750, 50) mm, rotated rx 180 ry 0 rz 90 deg; joints [-10.635, -71.942, 120.671, 165.972, 49.587, -170.8]
  MoveL 262 to (-389.22, 800, 50) mm, rotated rx 180 ry 0 rz 90 deg; joints [-11.008, -73.795, 123.356, 165.663, 50.454, -170.757]
  MoveL 263 to (-389.22, 800, -0.5) mm, rotated rx -180 ry 0 rz 90 deg; joints [-11.008, -71.329, 123.714, 166.203, 53.193, -171.63]
  MoveL 264 to (-389.22, 800, 50) mm, rotated rx 180 ry 0 rz 90 deg; joints [-11.008, -73.795, 123.356, 165.663, 50.454, -170.757]
  MoveL 265 to (-389.22, 850, 50) mm, rotated rx -180 ry 0 rz 90 deg; joints [-11.408, -75.674, 126.003, 165.311, 51.261, -170.684]
  MoveL 266 to (-389.22, 850, -0.5) mm, rotated rx -180 ry 0 rz 90 deg; joints [-11.408, -73.094, 126.374, 165.871, 54.12, -171.608]
  MoveL 267 to (-389.22, 850, 50) mm, rotated rx -180 ry 0 rz 90 deg; joints [-11.408, -75.674, 126.003, 165.311, 51.261, -170.684]
  MoveL 268 to (-389.22, 900, 50) mm, rotated rx 180 ry 0 rz 90 deg; joints [-11.837, -77.587, 128.614, 164.913, 52.006, -170.578]
  MoveL 269 to (-389.22, 900, -0.5) mm, rotated rx -180 ry 0 rz 90 deg; joints [-11.837, -74.881, 128.999, 165.497, 54.994, -171.559]
  MoveL 270 to (-389.22, 900, 50) mm, rotated rx 180 ry 0 rz 90 deg; joints [-11.837, -77.587, 128.614, 164.913, 52.006, -170.578]
  MoveL 271 to (-389.22, 950, 50) mm, rotated rx -180 ry 0 rz 90 deg; joints [-12.299, -79.542, 131.19, 164.464, 52.681, -170.433]
  MoveL 272 to (-389.22, 950, -0.5) mm, rotated rx -180 ry 0 rz 90 deg; joints [-12.299, -76.7, 131.591, 165.077, 55.811, -171.483]
  MoveL 273 to (-389.22, 950, 50) mm, rotated rx -180 ry 0 rz 90 deg; joints [-12.299, -79.542, 131.19, 164.464, 52.681, -170.433]
  MoveL 274 to (-389.22, 1000, 50) mm, rotated rx 180 ry 0 rz 90 deg; joints [-12.798, -81.549, 133.733, 163.957, 53.28, -170.244]
  MoveL 275 to (-389.22, 1000, -0.5) mm, rotated rx 180 ry 0 rz 90 deg; joints [-12.798, -78.557, 134.152, 164.606, 56.564, -171.374]
  MoveL 276 to (-389.22, 1000, 50) mm, rotated rx 180 ry 0 rz 90 deg; joints [-12.798, -81.549, 133.733, 163.957, 53.28, -170.244]
  MoveL 277 to (-389.22, 1050, 50) mm, rotated rx 180 ry 0 rz 90 deg; joints [-13.339, -83.621, 136.244, 163.386, 53.795, -170.004]
  MoveL 278 to (-389.22, 1050, -0.5) mm, rotated rx 180 ry 0 rz 90 deg; joints [-13.339, -80.463, 136.683, 164.078, 57.248, -171.227]
  MoveL 279 to (-389.22, 1050, 50) mm, rotated rx 180 ry 0 rz 90 deg; joints [-13.339, -83.621, 136.244, 163.386, 53.795, -170.004]
  MoveL 280 to (-389.22, 1100, 50) mm, rotated rx 180 ry 0 rz 90 deg; joints [-13.927, -85.77, 138.723, 162.741, 54.214, -169.703]
  MoveL 281 to (-389.22, 1100, -0.5) mm, rotated rx -180 ry 0 rz 90 deg; joints [-13.927, -82.43, 139.185, 163.485, 57.852, -171.035]
  MoveL 282 to (-389.22, 1100, 50) mm, rotated rx 180 ry 0 rz 90 deg; joints [-13.927, -85.77, 138.723, 162.741, 54.214, -169.703]
  MoveL 283 to (-389.22, 1150, 50) mm, rotated rx 180 ry 0 rz 90 deg; joints [-14.567, -88.014, 141.17, 162.01, 54.524, -169.327]
  MoveL 284 to (-389.22, 1150, -0.5) mm, rotated rx 180 ry 0 rz 90 deg; joints [-14.567, -84.472, 141.659, 162.818, 58.367, -170.789]
  MoveL 285 to (-389.22, 1150, 50) mm, rotated rx 180 ry 0 rz 90 deg; joints [-14.567, -88.014, 141.17, 162.01, 54.524, -169.327]
  MoveL 286 to (-389.22, 1200, 50) mm, rotated rx 180 ry 0 rz 90 deg; joints [-15.268, -90.374, 143.586, 161.179, 54.709, -168.86]
  MoveL 287 to (-389.22, 1200, -0.5) mm, rotated rx -180 ry 0 rz 90 deg; joints [-15.268, -86.606, 144.104, 162.066, 58.778, -170.476]
  MoveL 288 to (-389.22, 1200, 50) mm, rotated rx 180 ry 0 rz 90 deg; joints [-15.268, -90.374, 143.586, 161.179, 54.709, -168.86]
  MoveL 289 to (-389.22, 1250, 50) mm, rotated rx -180 ry 0 rz 90 deg; joints [-16.037, -92.876, 145.969, 160.227, 54.75, -168.279]
  MoveL 290 to (-389.22, 1250, -0.5) mm, rotated rx -180 ry 0 rz 90 deg; joints [-16.037, -88.855, 146.522, 161.212, 59.068, -170.081]
  MoveL 291 to (-389.22, 1250, 50) mm, rotated rx -180 ry 0 rz 90 deg; joints [-16.037, -92.876, 145.969, 160.227, 54.75, -168.279]
  MoveL 292 to (-48.6, 1150, 50) mm, rotated rx 180 ry 0 rz 90 deg; joints [-30.403, -82.147, 134.47, 143.448, 58.186, -158.653]
  MoveL 293 to (-48.6, 1150, -0.5) mm, rotated rx -180 ry 0 rz 90 deg; joints [-30.403, -79.109, 134.895, 144.642, 60.99, -161.011]
  MoveL 294 to (-48.6, 1150, 50) mm, rotated rx 180 ry 0 rz 90 deg; joints [-30.403, -82.147, 134.47, 143.448, 58.186, -158.653]
  MoveL 295 to (-103.93, 1150, 50) mm, rotated rx 180 ry 0 rz 90 deg; joints [-28.087, -83.3, 135.863, 146.095, 57.568, -160.178]
  MoveL 296 to (-103.93, 1150, -0.5) mm, rotated rx -180 ry 0 rz 90 deg; joints [-28.087, -80.169, 136.299, 147.27, 60.549, -162.463]
  MoveL 297 to (-103.93, 1150, 50) mm, rotated rx 180 ry 0 rz 90 deg; joints [-28.087, -83.3, 135.863, 146.095, 57.568, -160.178]
  MoveL 298 to (-174.73, 1150, 50) mm, rotated rx 180 ry 0 rz 90 deg; joints [-24.972, -84.68, 137.482, 149.687, 56.766, -162.233]
  MoveL 299 to (-174.73, 1150, -0.5) mm, rotated rx -180 ry 0 rz 90 deg; joints [-24.972, -81.434, 137.932, 150.817, 59.976, -164.387]
  MoveL 300 to (-174.73, 1150, 50) mm, rotated rx 180 ry 0 rz 90 deg; joints [-24.972, -84.68, 137.482, 149.687, 56.766, -162.233]
  MoveL 301 to (-230.06, 1150, 50) mm, rotated rx 180 ry 0 rz 90 deg; joints [-22.422, -85.673, 138.614, 152.659, 56.146, -163.932]
  MoveL 302 to (-230.06, 1150, -0.5) mm, rotated rx -180 ry 0 rz 90 deg; joints [-22.422, -82.342, 139.075, 153.735, 59.531, -165.952]
  MoveL 303 to (-230.06, 1150, 50) mm, rotated rx 180 ry 0 rz 90 deg; joints [-22.422, -85.673, 138.614, 152.659, 56.146, -163.932]
  MoveL 304 to (-300.86, 1150, 50) mm, rotated rx 180 ry 0 rz 90 deg; joints [-19.017, -86.817, 139.883, 156.675, 55.382, -166.236]
  MoveL 305 to (-300.86, 1150, -0.5) mm, rotated rx 180 ry 0 rz 90 deg; joints [-19.017, -83.384, 140.357, 157.653, 58.983, -168.04]
  MoveL 306 to (-300.86, 1150, 50) mm, rotated rx 180 ry 0 rz 90 deg; joints [-19.017, -86.817, 139.883, 156.675, 55.382, -166.236]
  MoveL 307 to (-356.19, 1150, 50) mm, rotated rx -180 ry 0 rz 90 deg; joints [-16.255, -87.599, 140.729, 159.975, 54.828, -168.144]
  MoveL 308 to (-356.19, 1150, -0.5) mm, rotated rx 180 ry 0 rz 90 deg; joints [-16.255, -84.095, 141.212, 160.853, 58.586, -169.743]
  MoveL 309 to (-356.19, 1150, 50) mm, rotated rx -180 ry 0 rz 90 deg; joints [-16.255, -87.599, 140.729, 159.975, 54.828, -168.144]
  MoveL 310 to (-450.8, 300, 50) mm, rotated rx 180 ry 0 rz 90 deg; joints [-6.31, -55.796, 94.774, 170.03, 39.405, -172.265]
  MoveL 311 to (-450.8, 300, -0.5) mm, rotated rx 180 ry 0 rz 90 deg; joints [-6.31, -54.103, 95.068, 170.427, 41.363, -172.786]
  MoveL 312 to (-450.8, 300, 50) mm, rotated rx 180 ry 0 rz 90 deg; joints [-6.31, -55.796, 94.774, 170.03, 39.405, -172.265]
  MoveL 313 to (-450.8, 350, 50) mm, rotated rx 180 ry 0 rz 90 deg; joints [-6.479, -57.668, 97.96, 170.039, 40.722, -172.419]
  MoveL 314 to (-450.8, 350, -0.5) mm, rotated rx -180 ry 0 rz 90 deg; joints [-6.479, -55.916, 98.256, 170.429, 42.741, -172.94]
  MoveL 315 to (-450.8, 350, 50) mm, rotated rx 180 ry 0 rz 90 deg; joints [-6.479, -57.668, 97.96, 170.039, 40.722, -172.419]
  MoveL 316 to (-450.8, 400, 50) mm, rotated rx -180 ry 0 rz 90 deg; joints [-6.659, -59.518, 101.071, 170.018, 41.987, -172.547]
  MoveL 317 to (-450.8, 400, -0.5) mm, rotated rx -180 ry 0 rz 90 deg; joints [-6.659, -57.705, 101.371, 170.403, 44.069, -173.073]
  MoveL 318 to (-450.8, 400, 50) mm, rotated rx -180 ry 0 rz 90 deg; joints [-6.659, -59.518, 101.071, 170.018, 41.987, -172.547]
  MoveL 319 to (-450.8, 450, 50) mm, rotated rx 180 ry 0 rz 90 deg; joints [-6.848, -61.353, 104.114, 169.969, 43.201, -172.653]
  MoveL 320 to (-450.8, 450, -0.5) mm, rotated rx 180 ry 0 rz 90 deg; joints [-6.848, -59.474, 104.418, 170.352, 45.352, -173.187]
  MoveL 321 to (-450.8, 450, 50) mm, rotated rx 180 ry 0 rz 90 deg; joints [-6.848, -61.353, 104.114, 169.969, 43.201, -172.653]
  MoveL 322 to (-450.8, 500, 50) mm, rotated rx 180 ry 0 rz 90 deg; joints [-7.048, -63.178, 107.095, 169.893, 44.365, -172.738]
  MoveL 323 to (-450.8, 500, -0.5) mm, rotated rx 180 ry 0 rz 90 deg; joints [-7.048, -61.229, 107.404, 170.275, 46.589, -173.283]
  MoveL 324 to (-450.8, 500, 50) mm, rotated rx 180 ry 0 rz 90 deg; joints [-7.048, -63.178, 107.095, 169.893, 44.365, -172.738]
  MoveL 325 to (-450.8, 550, 50) mm, rotated rx -180 ry 0 rz 90 deg; joints [-7.261, -64.997, 110.019, 169.79, 45.479, -172.802]
  MoveL 326 to (-450.8, 550, -0.5) mm, rotated rx 180 ry 0 rz 90 deg; joints [-7.261, -62.974, 110.333, 170.174, 47.781, -173.362]
  MoveL 327 to (-450.8, 550, 50) mm, rotated rx -180 ry 0 rz 90 deg; joints [-7.261, -64.997, 110.019, 169.79, 45.479, -172.802]
  MoveL 328 to (-450.8, 600, 50) mm, rotated rx -180 ry 0 rz 90 deg; joints [-7.486, -66.816, 112.89, 169.66, 46.543, -172.847]
  MoveL 329 to (-450.8, 600, -0.5) mm, rotated rx -180 ry 0 rz 90 deg; joints [-7.486, -64.712, 113.212, 170.048, 48.93, -173.424]
  MoveL 330 to (-450.8, 600, 50) mm, rotated rx -180 ry 0 rz 90 deg; joints [-7.486, -66.816, 112.89, 169.66, 46.543, -172.847]
  MoveL 331 to (-450.8, 650, 50) mm, rotated rx -180 ry 0 rz 90 deg; joints [-7.726, -68.639, 115.713, 169.503, 47.556, -172.873]
  MoveL 332 to (-450.8, 650, -0.5) mm, rotated rx -180 ry 0 rz 90 deg; joints [-7.726, -66.45, 116.042, 169.898, 50.034, -173.471]
  MoveL 333 to (-450.8, 650, 50) mm, rotated rx -180 ry 0 rz 90 deg; joints [-7.726, -68.639, 115.713, 169.503, 47.556, -172.873]
  MoveL 334 to (-450.8, 700, 50) mm, rotated rx 180 ry 0 rz 90 deg; joints [-7.982, -70.472, 118.491, 169.318, 48.516, -172.878]
  MoveL 335 to (-450.8, 700, -0.5) mm, rotated rx -180 ry 0 rz 90 deg; joints [-7.982, -68.191, 118.829, 169.721, 51.092, -173.502]
  MoveL 336 to (-450.8, 700, 50) mm, rotated rx 180 ry 0 rz 90 deg; joints [-7.982, -70.472, 118.491, 169.318, 48.516, -172.878]
  MoveL 337 to (-450.8, 750, 50) mm, rotated rx -180 ry 0 rz 90 deg; joints [-8.255, -72.322, 121.227, 169.104, 49.421, -172.862]
  MoveL 338 to (-450.8, 750, -0.5) mm, rotated rx -180 ry 0 rz 90 deg; joints [-8.255, -69.941, 121.576, 169.517, 52.104, -173.516]
  MoveL 339 to (-450.8, 750, 50) mm, rotated rx -180 ry 0 rz 90 deg; joints [-8.255, -72.322, 121.227, 169.104, 49.421, -172.862]
  MoveL 340 to (-450.8, 800, 50) mm, rotated rx 180 ry 0 rz 90 deg; joints [-8.547, -74.193, 123.924, 168.857, 50.267, -172.824]
  MoveL 341 to (-450.8, 800, -0.5) mm, rotated rx -180 ry 0 rz 90 deg; joints [-8.547, -71.704, 124.284, 169.285, 53.066, -173.513]
  MoveL 342 to (-450.8, 800, 50) mm, rotated rx 180 ry 0 rz 90 deg; joints [-8.547, -74.193, 123.924, 168.857, 50.267, -172.824]
  MoveL 343 to (-450.8, 850, 50) mm, rotated rx -180 ry 0 rz 90 deg; joints [-8.86, -76.094, 126.584, 168.577, 51.051, -172.761]
  MoveL 344 to (-450.8, 850, -0.5) mm, rotated rx 180 ry 0 rz 90 deg; joints [-8.86, -73.487, 126.957, 169.021, 53.975, -173.491]
  MoveL 345 to (-450.8, 850, 50) mm, rotated rx -180 ry 0 rz 90 deg; joints [-8.86, -76.094, 126.584, 168.577, 51.051, -172.761]
  MoveL 346 to (-450.8, 900, 50) mm, rotated rx -180 ry 0 rz 90 deg; joints [-9.197, -78.032, 129.209, 168.259, 51.767, -172.671]
  MoveL 347 to (-450.8, 900, -0.5) mm, rotated rx -180 ry 0 rz 90 deg; joints [-9.197, -75.296, 129.597, 168.724, 54.829, -173.448]
  MoveL 348 to (-450.8, 900, 50) mm, rotated rx -180 ry 0 rz 90 deg; joints [-9.197, -78.032, 129.209, 168.259, 51.767, -172.671]
  MoveL 349 to (-450.8, 950, 50) mm, rotated rx -180 ry 0 rz 90 deg; joints [-9.561, -80.017, 131.801, 167.9, 52.408, -172.549]
  MoveL 350 to (-450.8, 950, -0.5) mm, rotated rx 180 ry 0 rz 90 deg; joints [-9.561, -77.14, 132.206, 168.39, 55.62, -173.382]
  MoveL 351 to (-450.8, 950, 50) mm, rotated rx -180 ry 0 rz 90 deg; joints [-9.561, -80.017, 131.801, 167.9, 52.408, -172.549]
  MoveL 352 to (-450.8, 1000, 50) mm, rotated rx 180 ry 0 rz 90 deg; joints [-9.954, -82.059, 134.362, 167.494, 52.966, -172.391]
  MoveL 353 to (-450.8, 1000, -0.5) mm, rotated rx 180 ry 0 rz 90 deg; joints [-9.954, -79.027, 134.786, 168.014, 56.343, -173.289]
  MoveL 354 to (-450.8, 1000, 50) mm, rotated rx 180 ry 0 rz 90 deg; joints [-9.954, -82.059, 134.362, 167.494, 52.966, -172.391]
  MoveL 355 to (-450.8, 1050, 50) mm, rotated rx 180 ry 0 rz 90 deg; joints [-10.381, -84.172, 136.892, 167.035, 53.431, -172.19]
  MoveL 356 to (-450.8, 1050, -0.5) mm, rotated rx 180 ry 0 rz 90 deg; joints [-10.381, -80.969, 137.337, 167.592, 56.99, -173.165]
  MoveL 357 to (-450.8, 1050, 50) mm, rotated rx 180 ry 0 rz 90 deg; joints [-10.381, -84.172, 136.892, 167.035, 53.431, -172.19]
  MoveL 358 to (-450.8, 1100, 50) mm, rotated rx 180 ry 0 rz 90 deg; joints [-10.845, -86.371, 139.392, 166.515, 53.788, -171.936]
  MoveL 359 to (-450.8, 1100, -0.5) mm, rotated rx 180 ry 0 rz 90 deg; joints [-10.845, -82.978, 139.862, 167.116, 57.549, -173.003]
  MoveL 360 to (-450.8, 1100, 50) mm, rotated rx 180 ry 0 rz 90 deg; joints [-10.845, -86.371, 139.392, 166.515, 53.788, -171.936]
  MoveL 361 to (-450.8, 1150, 50) mm, rotated rx 180 ry 0 rz 90 deg; joints [-11.352, -88.675, 141.863, 165.922, 54.022, -171.619]
  MoveL 362 to (-450.8, 1150, -0.5) mm, rotated rx 180 ry 0 rz 90 deg; joints [-11.352, -85.071, 142.36, 166.58, 58.006, -172.795]
  MoveL 363 to (-450.8, 1150, 50) mm, rotated rx 180 ry 0 rz 90 deg; joints [-11.352, -88.675, 141.863, 165.922, 54.022, -171.619]
  MoveL 364 to (-450.8, 1200, 50) mm, rotated rx -180 ry 0 rz 90 deg; joints [-11.908, -91.109, 144.304, 165.244, 54.113, -171.223]
  MoveL 365 to (-450.8, 1200, -0.5) mm, rotated rx 180 ry 0 rz 90 deg; joints [-11.908, -87.268, 144.833, 165.971, 58.345, -172.53]
  MoveL 366 to (-450.8, 1200, 50) mm, rotated rx -180 ry 0 rz 90 deg; joints [-11.908, -91.109, 144.304, 165.244, 54.113, -171.223]
  MoveL 367 to (-450.8, 1250, 50) mm, rotated rx -180 ry 0 rz 90 deg; joints [-12.521, -93.702, 146.716, 164.463, 54.033, -170.726]
  MoveL 368 to (-450.8, 1250, -0.5) mm, rotated rx 180 ry 0 rz 90 deg; joints [-12.521, -89.595, 147.281, 165.277, 58.544, -172.192]
  MoveL 369 to (-450.8, 1250, 50) mm, rotated rx -180 ry 0 rz 90 deg; joints [-12.521, -93.702, 146.716, 164.463, 54.033, -170.726]
  MoveL 370 to (-450.8, 1300, 50) mm, rotated rx -180 ry 0 rz 90 deg; joints [-13.199, -96.493, 149.095, 163.553, 53.75, -170.098]
  MoveL 371 to (-450.8, 1300, -0.5) mm, rotated rx 180 ry 0 rz 90 deg; joints [-13.199, -92.087, 149.703, 164.479, 58.571, -171.76]
  MoveL 372 to (-450.8, 1300, 50) mm, rotated rx -180 ry 0 rz 90 deg; joints [-13.199, -96.493, 149.095, 163.553, 53.75, -170.098]
  MoveL 373 to (-450.8, 1350, 50) mm, rotated rx -180 ry 0 rz 90 deg; joints [-13.953, -99.532, 151.44, 162.48, 53.222, -169.297]
  MoveL 374 to (-450.8, 1350, -0.5) mm, rotated rx -180 ry 0 rz 90 deg; joints [-13.953, -94.787, 152.099, 163.553, 58.39, -171.204]
  MoveL 375 to (-450.8, 1350, 50) mm, rotated rx -180 ry 0 rz 90 deg; joints [-13.953, -99.532, 151.44, 162.48, 53.222, -169.297]
  MoveL 376 to (-450.8, 1400, 50) mm, rotated rx -180 ry 0 rz 90 deg; joints [-14.796, -102.885, 153.748, 161.194, 52.392, -168.26]
  MoveL 377 to (-450.8, 1400, -0.5) mm, rotated rx -180 ry 0 rz 90 deg; joints [-14.796, -97.758, 154.467, 162.463, 57.948, -170.48]
  MoveL 378 to (-450.8, 1400, 50) mm, rotated rx -180 ry 0 rz 90 deg; joints [-14.796, -102.885, 153.748, 161.194, 52.392, -168.26]
  MoveL 379 to (-450.8, 1450, 50) mm, rotated rx 180 ry 0 rz 70 deg; joints [-22.366, -102.67, 153.608, 130.41, 62.251, -151.326]
  MoveL 380 to (-450.8, 1450, -0.5) mm, rotated rx 180 ry 0 rz 70 deg; joints [-22.366, -97.567, 154.323, 132.521, 66.106, -156.169]
  MoveL 381 to (-450.8, 1450, 50) mm, rotated rx 180 ry 0 rz 70 deg; joints [-22.366, -102.67, 153.608, 130.41, 62.251, -151.326]
  MoveL 382 to (-829.2, 100, 50) mm, rotated rx -180 ry 0 rz 90 deg; joints [4.624, -48.13, 81.363, 188.395, 33.517, -187.014]
  MoveL 383 to (-829.2, 100, -0.5) mm, rotated rx -180 ry 0 rz 90 deg; joints [4.624, -46.638, 81.656, 188.023, 35.284, -186.563]
  MoveL 384 to (-829.2, 100, 50) mm, rotated rx 180 ry 0 rz 90 deg; joints [4.624, -48.13, 81.363, 188.395, 33.517, -187.014]
  MoveL 385 to (-829.2, 150, 50) mm, rotated rx -180 ry 0 rz 90 deg; joints [4.737, -50.146, 84.941, 188.262, 35.075, -186.777]
  MoveL 386 to (-829.2, 150, -0.5) mm, rotated rx 180 ry 0 rz 90 deg; joints [4.737, -48.607, 85.233, 187.907, 36.889, -186.339]
  MoveL 387 to (-829.2, 150, 50) mm, rotated rx -180 ry 0 rz 90 deg; joints [4.737, -50.146, 84.941, 188.262, 35.075, -186.777]
  MoveL 388 to (-829.2, 200, 50) mm, rotated rx -180 ry 0 rz 90 deg; joints [4.855, -52.116, 88.404, 188.167, 36.566, -186.575]
  MoveL 389 to (-829.2, 200, -0.5) mm, rotated rx 180 ry 0 rz 90 deg; joints [4.855, -50.527, 88.695, 187.826, 38.429, -186.146]
  MoveL 390 to (-829.2, 200, 50) mm, rotated rx -180 ry 0 rz 90 deg; joints [4.855, -52.116, 88.404, 188.167, 36.566, -186.575]
  MoveL 391 to (-829.2, 250, 50) mm, rotated rx 180 ry 0 rz 90 deg; joints [4.979, -54.048, 91.764, 188.106, 37.995, -186.404]
  MoveL 392 to (-829.2, 250, -0.5) mm, rotated rx 180 ry 0 rz 90 deg; joints [4.979, -52.405, 92.056, 187.775, 39.911, -185.979]
  MoveL 393 to (-829.2, 250, 50) mm, rotated rx 180 ry 0 rz 90 deg; joints [4.979, -54.048, 91.764, 188.106, 37.995, -186.404]
  MoveL 394 to (-829.2, 300, 50) mm, rotated rx -180 ry 0 rz 90 deg; joints [5.11, -55.947, 95.033, 188.073, 39.365, -186.258]
  MoveL 395 to (-829.2, 300, -0.5) mm, rotated rx 180 ry 0 rz 90 deg; joints [5.11, -54.249, 95.326, 187.75, 41.338, -185.835]
  MoveL 396 to (-829.2, 300, 50) mm, rotated rx -180 ry 0 rz 90 deg; joints [5.11, -55.947, 95.033, 188.073, 39.365, -186.258]
  MoveL 397 to (-829.2, 350, 50) mm, rotated rx 180 ry 0 rz 90 deg; joints [5.248, -57.821, 98.219, 188.067, 40.68, -186.135]
  MoveL 398 to (-829.2, 350, -0.5) mm, rotated rx -180 ry 0 rz 90 deg; joints [5.248, -56.064, 98.515, 187.75, 42.713, -185.71]
  MoveL 399 to (-829.2, 350, 50) mm, rotated rx 180 ry 0 rz 90 deg; joints [5.248, -57.821, 98.219, 188.067, 40.68, -186.135]
  MoveL 400 to (-829.2, 400, 50) mm, rotated rx -180 ry 0 rz 90 deg; joints [5.394, -59.674, 101.331, 188.085, 41.942, -186.032]
  MoveL 401 to (-829.2, 400, -0.5) mm, rotated rx -180 ry 0 rz 90 deg; joints [5.394, -57.855, 101.631, 187.772, 44.04, -185.603]
  MoveL 402 to (-829.2, 400, 50) mm, rotated rx -180 ry 0 rz 90 deg; joints [5.394, -59.674, 101.331, 188.085, 41.942, -186.032]
  MoveL 403 to (-829.2, 450, 50) mm, rotated rx 180 ry 0 rz 90 deg; joints [5.548, -61.512, 104.376, 188.126, 43.152, -185.947]
  MoveL 404 to (-829.2, 450, -0.5) mm, rotated rx 180 ry 0 rz 90 deg; joints [5.548, -59.627, 104.68, 187.814, 45.32, -185.512]
  MoveL 405 to (-829.2, 450, 50) mm, rotated rx 180 ry 0 rz 90 deg; joints [5.548, -61.512, 104.376, 188.126, 43.152, -185.947]
  MoveL 406 to (-829.2, 500, 50) mm, rotated rx 180 ry 0 rz 90 deg; joints [5.711, -63.341, 107.359, 188.189, 44.312, -185.879]
  MoveL 407 to (-829.2, 500, -0.5) mm, rotated rx -180 ry 0 rz 90 deg; joints [5.711, -61.386, 107.668, 187.877, 46.554, -185.435]
  MoveL 408 to (-829.2, 500, 50) mm, rotated rx 180 ry 0 rz 90 deg; joints [5.711, -63.341, 107.359, 188.189, 44.312, -185.879]
  MoveL 409 to (-829.2, 550, 50) mm, rotated rx -180 ry 0 rz 90 deg; joints [5.883, -65.165, 110.286, 188.274, 45.421, -185.828]
  MoveL 410 to (-829.2, 550, -0.5) mm, rotated rx -180 ry 0 rz 90 deg; joints [5.883, -63.134, 110.601, 187.961, 47.743, -185.372]
  MoveL 411 to (-829.2, 550, 50) mm, rotated rx -180 ry 0 rz 90 deg; joints [5.883, -65.165, 110.286, 188.274, 45.421, -185.828]
  MoveL 412 to (-829.2, 600, 50) mm, rotated rx 180 ry 0 rz 90 deg; joints [6.067, -66.989, 113.161, 188.381, 46.479, -185.793]
  MoveL 413 to (-829.2, 600, -0.5) mm, rotated rx -180 ry 0 rz 90 deg; joints [6.067, -64.878, 113.483, 188.064, 48.887, -185.322]
  MoveL 414 to (-829.2, 600, 50) mm, rotated rx 180 ry 0 rz 90 deg; joints [6.067, -66.989, 113.161, 188.381, 46.479, -185.793]
  MoveL 415 to (-829.2, 650, 50) mm, rotated rx 180 ry 0 rz 90 deg; joints [6.262, -68.819, 115.988, 188.51, 47.485, -185.774]
  MoveL 416 to (-829.2, 650, -0.5) mm, rotated rx 180 ry 0 rz 90 deg; joints [6.262, -66.621, 116.318, 188.187, 49.987, -185.285]
  MoveL 417 to (-829.2, 650, 50) mm, rotated rx 180 ry 0 rz 90 deg; joints [6.262, -68.819, 115.988, 188.51, 47.485, -185.774]
  MoveL 418 to (-829.2, 700, 50) mm, rotated rx 180 ry 0 rz 90 deg; joints [6.47, -70.66, 118.771, 188.662, 48.437, -185.771]
  MoveL 419 to (-829.2, 700, -0.5) mm, rotated rx 180 ry 0 rz 90 deg; joints [6.47, -68.368, 119.11, 188.332, 51.04, -185.262]
  MoveL 420 to (-829.2, 700, 50) mm, rotated rx 180 ry 0 rz 90 deg; joints [6.47, -70.66, 118.771, 188.662, 48.437, -185.771]
  MoveL 421 to (-829.2, 750, 50) mm, rotated rx 180 ry 0 rz 90 deg; joints [6.692, -72.517, 121.512, 188.838, 49.333, -185.786]
  MoveL 422 to (-829.2, 750, -0.5) mm, rotated rx 180 ry 0 rz 90 deg; joints [6.692, -70.125, 121.862, 188.499, 52.044, -185.251]
  MoveL 423 to (-829.2, 750, 50) mm, rotated rx 180 ry 0 rz 90 deg; joints [6.692, -72.517, 121.512, 188.838, 49.333, -185.786]
  MoveL 424 to (-829.2, 800, 50) mm, rotated rx -180 ry 0 rz 90 deg; joints [6.93, -74.399, 124.215, 189.04, 50.169, -185.819]
  MoveL 425 to (-829.2, 800, -0.5) mm, rotated rx 180 ry 0 rz 90 deg; joints [6.93, -71.897, 124.577, 188.69, 52.999, -185.256]
  MoveL 426 to (-829.2, 800, 50) mm, rotated rx -180 ry 0 rz 90 deg; joints [6.93, -74.399, 124.215, 189.04, 50.169, -185.819]
  MoveL 427 to (-829.2, 850, 50) mm, rotated rx -180 ry 0 rz 90 deg; joints [7.186, -76.311, 126.882, 189.271, 50.94, -185.873]
  MoveL 428 to (-829.2, 850, -0.5) mm, rotated rx 180 ry 0 rz 90 deg; joints [7.186, -73.69, 127.257, 188.906, 53.899, -185.275]
  MoveL 429 to (-829.2, 850, 50) mm, rotated rx -180 ry 0 rz 90 deg; joints [7.186, -76.311, 126.882, 189.271, 50.94, -185.873]
  MoveL 430 to (-829.2, 900, 50) mm, rotated rx -180 ry 0 rz 90 deg; joints [7.461, -78.263, 129.515, 189.532, 51.641, -185.949]
  MoveL 431 to (-829.2, 900, -0.5) mm, rotated rx -180 ry 0 rz 90 deg; joints [7.461, -75.511, 129.905, 189.15, 54.741, -185.312]
  MoveL 432 to (-829.2, 900, 50) mm, rotated rx -180 ry 0 rz 90 deg; joints [7.461, -78.263, 129.515, 189.532, 51.641, -185.949]
  MoveL 433 to (-829.2, 950, 50) mm, rotated rx -180 ry 0 rz 90 deg; joints [7.758, -80.263, 132.116, 189.828, 52.263, -186.052]
  MoveL 434 to (-829.2, 950, -0.5) mm, rotated rx -180 ry 0 rz 90 deg; joints [7.758, -77.368, 132.523, 189.425, 55.519, -185.369]
  MoveL 435 to (-829.2, 950, 50) mm, rotated rx -180 ry 0 rz 90 deg; joints [7.758, -80.263, 132.116, 189.828, 52.263, -186.052]
  MoveL 436 to (-829.2, 1000, 50) mm, rotated rx 180 ry 0 rz 90 deg; joints [8.079, -82.324, 134.686, 190.162, 52.799, -186.185]
  MoveL 437 to (-829.2, 1000, -0.5) mm, rotated rx 180 ry 0 rz 90 deg; joints [8.079, -79.271, 135.112, 189.734, 56.226, -185.447]
  MoveL 438 to (-829.2, 1000, 50) mm, rotated rx 180 ry 0 rz 90 deg; joints [8.079, -82.324, 134.686, 190.162, 52.799, -186.185]
  MoveL 439 to (-829.2, 1050, 50) mm, rotated rx 180 ry 0 rz 90 deg; joints [8.428, -84.459, 137.226, 190.542, 53.236, -186.355]
  MoveL 440 to (-829.2, 1050, -0.5) mm, rotated rx -180 ry 0 rz 90 deg; joints [8.428, -81.232, 137.674, 190.081, 56.852, -185.553]
  MoveL 441 to (-829.2, 1050, 50) mm, rotated rx 180 ry 0 rz 90 deg; joints [8.428, -84.459, 137.226, 190.542, 53.236, -186.355]
  MoveL 442 to (-829.2, 1100, 50) mm, rotated rx -180 ry 0 rz 90 deg; joints [8.808, -86.685, 139.738, 190.972, 53.56, -186.569]
  MoveL 443 to (-829.2, 1100, -0.5) mm, rotated rx -180 ry 0 rz 90 deg; joints [8.808, -83.264, 140.211, 190.474, 57.385, -185.69]
  MoveL 444 to (-829.2, 1100, 50) mm, rotated rx -180 ry 0 rz 90 deg; joints [8.808, -86.685, 139.738, 190.972, 53.56, -186.569]
  MoveL 445 to (-829.2, 1150, 50) mm, rotated rx -180 ry 0 rz 90 deg; joints [9.223, -89.021, 142.221, 191.464, 53.752, -186.838]
  MoveL 446 to (-829.2, 1150, -0.5) mm, rotated rx 180 ry 0 rz 90 deg; joints [9.223, -85.384, 142.722, 190.917, 57.812, -185.866]
  MoveL 447 to (-829.2, 1150, 50) mm, rotated rx -180 ry 0 rz 90 deg; joints [9.223, -89.021, 142.221, 191.464, 53.752, -186.838]
  MoveL 448 to (-829.2, 1200, 50) mm, rotated rx -180 ry 0 rz 90 deg; joints [9.679, -91.495, 144.676, 192.028, 53.789, -187.174]
  MoveL 449 to (-829.2, 1200, -0.5) mm, rotated rx -180 ry 0 rz 90 deg; joints [9.679, -87.615, 145.21, 191.421, 58.111, -186.092]
  MoveL 450 to (-829.2, 1200, 50) mm, rotated rx -180 ry 0 rz 90 deg; joints [9.679, -91.495, 144.676, 192.028, 53.789, -187.174]
  MoveL 451 to (-829.2, 1250, 50) mm, rotated rx 180 ry 0 rz 90 deg; joints [10.183, -94.138, 147.102, 192.681, 53.642, -187.598]
  MoveL 452 to (-829.2, 1250, -0.5) mm, rotated rx -180 ry 0 rz 90 deg; joints [10.183, -89.985, 147.674, 191.998, 58.257, -186.38]
  MoveL 453 to (-829.2, 1250, 50) mm, rotated rx 180 ry 0 rz 90 deg; joints [10.183, -94.138, 147.102, 192.681, 53.642, -187.598]
  MoveL 454 to (-488.6, 1150, 50) mm, rotated rx -180 ry 0 rz 90 deg; joints [-9.341, -89.004, 142.203, 168.391, 53.765, -173.077]
  MoveL 455 to (-488.6, 1150, -0.5) mm, rotated rx -180 ry 0 rz 90 deg; joints [-9.341, -85.368, 142.704, 168.944, 57.821, -174.059]
  MoveL 456 to (-488.6, 1150, 50) mm, rotated rx -180 ry 0 rz 90 deg; joints [-9.341, -89.004, 142.203, 168.391, 53.765, -173.077]
  MoveL 457 to (-538.6, 1150, 50) mm, rotated rx 180 ry 0 rz 90 deg; joints [-6.645, -89.344, 142.551, 171.722, 53.495, -175.053]
  MoveL 458 to (-538.6, 1150, -0.5) mm, rotated rx 180 ry 0 rz 90 deg; joints [-6.645, -85.676, 143.056, 172.125, 57.627, -175.764]
  MoveL 459 to (-538.6, 1150, 50) mm, rotated rx 180 ry 0 rz 90 deg; joints [-6.645, -89.344, 142.551, 171.722, 53.495, -175.053]
  MoveL 460 to (-588.6, 1150, 50) mm, rotated rx -180 ry 0 rz 90 deg; joints [-3.92, -89.57, 142.781, 175.11, 53.311, -177.074]
  MoveL 461 to (-588.6, 1150, -0.5) mm, rotated rx -180 ry 0 rz 90 deg; joints [-3.92, -85.88, 143.289, 175.35, 57.495, -177.498]
  MoveL 462 to (-588.6, 1150, 50) mm, rotated rx -180 ry 0 rz 90 deg; joints [-3.92, -89.57, 142.781, 175.11, 53.311, -177.074]
  MoveL 463 to (-638.6, 1150, 50) mm, rotated rx 180 ry 0 rz 90 deg; joints [-1.177, -89.68, 142.892, 178.531, 53.221, -179.12]
  MoveL 464 to (-638.6, 1150, -0.5) mm, rotated rx 180 ry 0 rz 90 deg; joints [-1.177, -85.979, 143.401, 178.604, 57.43, -179.248]
  MoveL 465 to (-638.6, 1150, 50) mm, rotated rx 180 ry 0 rz 90 deg; joints [-1.177, -89.68, 142.892, 178.531, 53.221, -179.12]
  MoveL 466 to (-688.6, 1150, 50) mm, rotated rx -180 ry 0 rz 90 deg; joints [1.572, -89.671, 142.883, 181.963, 53.228, -181.175]
  MoveL 467 to (-688.6, 1150, -0.5) mm, rotated rx 180 ry 0 rz 90 deg; joints [1.572, -85.972, 143.393, 181.866, 57.435, -181.004]
  MoveL 468 to (-688.6, 1150, 50) mm, rotated rx -180 ry 0 rz 90 deg; joints [1.572, -89.671, 142.883, 181.963, 53.228, -181.175]
  MoveL 469 to (-738.6, 1150, 50) mm, rotated rx -180 ry 0 rz 90 deg; joints [4.314, -89.544, 142.755, 185.381, 53.332, -183.219]
  MoveL 470 to (-738.6, 1150, -0.5) mm, rotated rx 180 ry 0 rz 90 deg; joints [4.314, -85.857, 143.263, 185.116, 57.51, -182.753]
  MoveL 471 to (-738.6, 1150, 50) mm, rotated rx -180 ry 0 rz 90 deg; joints [4.314, -89.544, 142.755, 185.381, 53.332, -183.219]
  MoveL 472 to (-788.6, 1150, 50) mm, rotated rx 180 ry 0 rz 90 deg; joints [7.036, -89.302, 142.508, 188.761, 53.528, -185.234]
  MoveL 473 to (-788.6, 1150, -0.5) mm, rotated rx 180 ry 0 rz 90 deg; joints [7.036, -85.638, 143.013, 188.337, 57.651, -184.483]
  MoveL 474 to (-788.6, 1150, 50) mm, rotated rx 180 ry 0 rz 90 deg; joints [7.036, -89.302, 142.508, 188.761, 53.528, -185.234]
  MoveL 475 to (-890, 50, 50) mm, rotated rx 180 ry 0 rz 90 deg; joints [6.129, -45.818, 77.224, 191.643, 31.938, -189.919]
  MoveL 476 to (-890, 50, -0.5) mm, rotated rx -180 ry 0 rz 90 deg; joints [6.129, -44.378, 77.52, 191.111, 33.641, -189.286]
  MoveL 477 to (-890, 50, 50) mm, rotated rx 180 ry 0 rz 90 deg; joints [6.129, -45.818, 77.224, 191.643, 31.938, -189.919]
  MoveL 478 to (-890, 100, 50) mm, rotated rx 180 ry 0 rz 90 deg; joints [6.274, -47.892, 80.94, 191.398, 33.571, -189.535]
  MoveL 479 to (-890, 100, -0.5) mm, rotated rx 180 ry 0 rz 90 deg; joints [6.274, -46.406, 81.234, 190.897, 35.318, -188.927]
  MoveL 480 to (-890, 100, 50) mm, rotated rx 180 ry 0 rz 90 deg; joints [6.274, -47.892, 80.94, 191.398, 33.571, -189.535]
  MoveL 481 to (-890, 150, 50) mm, rotated rx -180 ry 0 rz 90 deg; joints [6.426, -49.91, 84.523, 191.216, 35.131, -189.211]
  MoveL 482 to (-890, 150, -0.5) mm, rotated rx 180 ry 0 rz 90 deg; joints [6.426, -48.376, 84.815, 190.738, 36.924, -188.62]
  MoveL 483 to (-890, 150, 50) mm, rotated rx -180 ry 0 rz 90 deg; joints [6.426, -49.91, 84.523, 191.216, 35.131, -189.211]
  MoveL 484 to (-890, 200, 50) mm, rotated rx 180 ry 0 rz 90 deg; joints [6.586, -51.879, 87.988, 191.085, 36.624, -188.936]
  MoveL 485 to (-890, 200, -0.5) mm, rotated rx -180 ry 0 rz 90 deg; joints [6.586, -50.295, 88.28, 190.626, 38.466, -188.357]
  MoveL 486 to (-890, 200, 50) mm, rotated rx 180 ry 0 rz 90 deg; joints [6.586, -51.879, 87.988, 191.085, 36.624, -188.936]
  MoveL 487 to (-890, 250, 50) mm, rotated rx 180 ry 0 rz 90 deg; joints [6.754, -53.809, 91.35, 190.999, 38.056, -188.701]
  MoveL 488 to (-890, 250, -0.5) mm, rotated rx -180 ry 0 rz 90 deg; joints [6.754, -52.173, 91.642, 190.554, 39.95, -188.129]
  MoveL 489 to (-890, 250, 50) mm, rotated rx 180 ry 0 rz 90 deg; joints [6.754, -53.809, 91.35, 190.999, 38.056, -188.701]
  MoveL 490 to (-890, 300, 50) mm, rotated rx -180 ry 0 rz 90 deg; joints [6.931, -55.705, 94.619, 190.953, 39.429, -188.502]
  MoveL 491 to (-890, 300, -0.5) mm, rotated rx -180 ry 0 rz 90 deg; joints [6.931, -54.015, 94.912, 190.519, 41.379, -187.932]
  MoveL 492 to (-890, 300, 50) mm, rotated rx -180 ry 0 rz 90 deg; joints [6.931, -55.705, 94.619, 190.953, 39.429, -188.502]
  MoveL 493 to (-890, 350, 50) mm, rotated rx -180 ry 0 rz 90 deg; joints [7.117, -57.575, 97.804, 190.942, 40.748, -188.333]
  MoveL 494 to (-890, 350, -0.5) mm, rotated rx 180 ry 0 rz 90 deg; joints [7.117, -55.827, 98.1, 190.516, 42.757, -187.761]
  MoveL 495 to (-890, 350, 50) mm, rotated rx -180 ry 0 rz 90 deg; joints [7.117, -57.575, 97.804, 190.942, 40.748, -188.333]
  MoveL 496 to (-890, 400, 50) mm, rotated rx -180 ry 0 rz 90 deg; joints [7.314, -59.424, 100.914, 190.964, 42.015, -188.191]
  MoveL 497 to (-890, 400, -0.5) mm, rotated rx -180 ry 0 rz 90 deg; joints [7.314, -57.614, 101.214, 190.543, 44.087, -187.614]
  MoveL 498 to (-890, 400, 50) mm, rotated rx -180 ry 0 rz 90 deg; joints [7.314, -59.424, 100.914, 190.964, 42.015, -188.191]
  MoveL 499 to (-890, 450, 50) mm, rotated rx -180 ry 0 rz 90 deg; joints [7.521, -61.257, 103.956, 191.017, 43.23, -188.074]
  MoveL 500 to (-890, 450, -0.5) mm, rotated rx 180 ry 0 rz 90 deg; joints [7.521, -59.382, 104.26, 190.599, 45.371, -187.489]
  MoveL 501 to (-890, 450, 50) mm, rotated rx -180 ry 0 rz 90 deg; joints [7.521, -61.257, 103.956, 191.017, 43.23, -188.074]
  MoveL 502 to (-890, 500, 50) mm, rotated rx -180 ry 0 rz 90 deg; joints [7.741, -63.08, 106.935, 191.1, 44.397, -187.98]
  MoveL 503 to (-890, 500, -0.5) mm, rotated rx -180 ry 0 rz 90 deg; joints [7.741, -61.135, 107.244, 190.682, 46.609, -187.383]
  MoveL 504 to (-890, 500, 50) mm, rotated rx -180 ry 0 rz 90 deg; joints [7.741, -63.08, 106.935, 191.1, 44.397, -187.98]
  MoveL 505 to (-890, 550, 50) mm, rotated rx -180 ry 0 rz 90 deg; joints [7.974, -64.896, 109.857, 191.212, 45.514, -187.908]
  MoveL 506 to (-890, 550, -0.5) mm, rotated rx 180 ry 0 rz 90 deg; joints [7.974, -62.877, 110.172, 190.792, 47.804, -187.296]
  MoveL 507 to (-890, 550, 50) mm, rotated rx -180 ry 0 rz 90 deg; joints [7.974, -64.896, 109.857, 191.212, 45.514, -187.908]
  MoveL 508 to (-890, 600, 50) mm, rotated rx 180 ry 0 rz 90 deg; joints [8.221, -66.711, 112.727, 191.353, 46.581, -187.858]
  MoveL 509 to (-890, 600, -0.5) mm, rotated rx -180 ry 0 rz 90 deg; joints [8.221, -64.613, 113.048, 190.929, 48.955, -187.226]
  MoveL 510 to (-890, 600, 50) mm, rotated rx 180 ry 0 rz 90 deg; joints [8.221, -66.711, 112.727, 191.353, 46.581, -187.858]
  MoveL 511 to (-890, 650, 50) mm, rotated rx -180 ry 0 rz 90 deg; joints [8.484, -68.531, 115.547, 191.524, 47.598, -187.829]
  MoveL 512 to (-890, 650, -0.5) mm, rotated rx 180 ry 0 rz 90 deg; joints [8.484, -66.347, 115.876, 191.093, 50.062, -187.174]
  MoveL 513 to (-890, 650, 50) mm, rotated rx -180 ry 0 rz 90 deg; joints [8.484, -68.531, 115.547, 191.524, 47.598, -187.829]
  MoveL 514 to (-890, 700, 50) mm, rotated rx 180 ry 0 rz 90 deg; joints [8.763, -70.36, 118.322, 191.726, 48.562, -187.821]
  MoveL 515 to (-890, 700, -0.5) mm, rotated rx -180 ry 0 rz 90 deg; joints [8.763, -68.084, 118.66, 191.286, 51.124, -187.139]
  MoveL 516 to (-890, 700, 50) mm, rotated rx 180 ry 0 rz 90 deg; joints [8.763, -70.36, 118.322, 191.726, 48.562, -187.821]
  MoveL 517 to (-890, 750, 50) mm, rotated rx 180 ry 0 rz 90 deg; joints [9.062, -72.204, 121.055, 191.96, 49.473, -187.837]
  MoveL 518 to (-890, 750, -0.5) mm, rotated rx 180 ry 0 rz 90 deg; joints [9.062, -69.829, 121.403, 191.508, 52.139, -187.123]
  MoveL 519 to (-890, 750, 50) mm, rotated rx 180 ry 0 rz 90 deg; joints [9.062, -72.204, 121.055, 191.96, 49.473, -187.837]
  MoveL 520 to (-890, 800, 50) mm, rotated rx 180 ry 0 rz 90 deg; joints [9.382, -74.07, 123.748, 192.228, 50.326, -187.877]
  MoveL 521 to (-890, 800, -0.5) mm, rotated rx -180 ry 0 rz 90 deg; joints [9.382, -71.588, 124.108, 191.762, 53.106, -187.125]
  MoveL 522 to (-890, 800, 50) mm, rotated rx 180 ry 0 rz 90 deg; joints [9.382, -74.07, 123.748, 192.228, 50.326, -187.877]
  MoveL 523 to (-890, 850, 50) mm, rotated rx -180 ry 0 rz 90 deg; joints [9.725, -75.964, 126.404, 192.533, 51.117, -187.944]
  MoveL 524 to (-890, 850, -0.5) mm, rotated rx 180 ry 0 rz 90 deg; joints [9.725, -73.365, 126.777, 192.049, 54.021, -187.147]
  MoveL 525 to (-890, 850, 50) mm, rotated rx -180 ry 0 rz 90 deg; joints [9.725, -75.964, 126.404, 192.533, 51.117, -187.944]
  MoveL 526 to (-890, 900, 50) mm, rotated rx 180 ry 0 rz 90 deg; joints [10.094, -77.894, 129.025, 192.879, 51.842, -188.041]
  MoveL 527 to (-890, 900, -0.5) mm, rotated rx -180 ry 0 rz 90 deg; joints [10.094, -75.167, 129.412, 192.373, 54.881, -187.193]
  MoveL 528 to (-890, 900, 50) mm, rotated rx 180 ry 0 rz 90 deg; joints [10.094, -77.894, 129.025, 192.879, 51.842, -188.041]
  MoveL 529 to (-890, 950, 50) mm, rotated rx -180 ry 0 rz 90 deg; joints [10.491, -79.869, 131.612, 193.27, 52.494, -188.171]
  MoveL 530 to (-890, 950, -0.5) mm, rotated rx 180 ry 0 rz 90 deg; joints [10.491, -77.003, 132.016, 192.737, 55.68, -187.263]
  MoveL 531 to (-890, 950, 50) mm, rotated rx -180 ry 0 rz 90 deg; joints [10.491, -79.869, 131.612, 193.27, 52.494, -188.171]
  MoveL 532 to (-890, 1000, 50) mm, rotated rx 180 ry 0 rz 90 deg; joints [10.921, -81.901, 134.167, 193.711, 53.065, -188.341]
  MoveL 533 to (-890, 1000, -0.5) mm, rotated rx -180 ry 0 rz 90 deg; joints [10.921, -78.881, 134.589, 193.146, 56.413, -187.362]
  MoveL 534 to (-890, 1000, 50) mm, rotated rx 180 ry 0 rz 90 deg; joints [10.921, -81.901, 134.167, 193.711, 53.065, -188.341]
  MoveL 535 to (-890, 1050, 50) mm, rotated rx -180 ry 0 rz 90 deg; joints [11.387, -84, 136.691, 194.209, 53.545, -188.556]
  MoveL 536 to (-890, 1050, -0.5) mm, rotated rx 180 ry 0 rz 90 deg; joints [11.387, -80.812, 137.134, 193.605, 57.071, -187.495]
  MoveL 537 to (-890, 1050, 50) mm, rotated rx -180 ry 0 rz 90 deg; joints [11.387, -84, 136.691, 194.209, 53.545, -188.556]
  MoveL 538 to (-890, 1100, 50) mm, rotated rx -180 ry 0 rz 90 deg; joints [11.894, -86.184, 139.185, 194.774, 53.922, -188.828]
  MoveL 539 to (-890, 1100, -0.5) mm, rotated rx 180 ry 0 rz 90 deg; joints [11.894, -82.807, 139.652, 194.122, 57.644, -187.668]
  MoveL 540 to (-890, 1100, 50) mm, rotated rx -180 ry 0 rz 90 deg; joints [11.894, -86.184, 139.185, 194.774, 53.922, -188.828]
  MoveL 541 to (-890, 1150, 50) mm, rotated rx 180 ry 0 rz 90 deg; joints [12.447, -88.469, 141.648, 195.415, 54.181, -189.167]
  MoveL 542 to (-890, 1150, -0.5) mm, rotated rx -180 ry 0 rz 90 deg; joints [12.447, -84.884, 142.143, 194.704, 58.12, -187.891]
  MoveL 543 to (-890, 1150, 50) mm, rotated rx 180 ry 0 rz 90 deg; joints [12.447, -88.469, 141.648, 195.415, 54.181, -189.167]
  MoveL 544 to (-890, 1200, 50) mm, rotated rx -180 ry 0 rz 90 deg; joints [13.054, -90.879, 144.081, 196.148, 54.302, -189.59]
  MoveL 545 to (-890, 1200, -0.5) mm, rotated rx 180 ry 0 rz 90 deg; joints [13.054, -87.061, 144.607, 195.364, 58.483, -188.174]
  MoveL 546 to (-890, 1200, 50) mm, rotated rx -180 ry 0 rz 90 deg; joints [13.054, -90.879, 144.081, 196.148, 54.302, -189.59]
  MoveL 547 to (-960, 50, 50) mm, rotated rx 180 ry 0 rz 90 deg; joints [7.973, -45.453, 76.566, 195.165, 32.019, -192.942]
  MoveL 548 to (-960, 50, -0.5) mm, rotated rx -180 ry 0 rz 90 deg; joints [7.973, -44.021, 76.864, 194.48, 33.691, -192.127]
  MoveL 549 to (-960, 50, 50) mm, rotated rx 180 ry 0 rz 90 deg; joints [7.973, -45.453, 76.566, 195.165, 32.019, -192.942]
  MoveL 550 to (-960, 100, 50) mm, rotated rx -180 ry 0 rz 90 deg; joints [8.161, -47.53, 80.293, 194.842, 33.654, -192.439]
  MoveL 551 to (-960, 100, -0.5) mm, rotated rx 180 ry 0 rz 90 deg; joints [8.161, -46.052, 80.587, 194.196, 35.369, -191.655]
  MoveL 552 to (-960, 100, 50) mm, rotated rx -180 ry 0 rz 90 deg; joints [8.161, -47.53, 80.293, 194.842, 33.654, -192.439]
  MoveL 553 to (-960, 150, 50) mm, rotated rx -180 ry 0 rz 90 deg; joints [8.358, -49.548, 83.882, 194.6, 35.216, -192.014]
  MoveL 554 to (-960, 150, -0.5) mm, rotated rx 180 ry 0 rz 90 deg; joints [8.358, -48.023, 84.175, 193.984, 36.977, -191.252]
  MoveL 555 to (-960, 150, 50) mm, rotated rx -180 ry 0 rz 90 deg; joints [8.358, -49.548, 83.882, 194.6, 35.216, -192.014]
  MoveL 556 to (-960, 200, 50) mm, rotated rx 180 ry 0 rz 90 deg; joints [8.565, -51.516, 87.353, 194.426, 36.712, -191.652]
  MoveL 557 to (-960, 200, -0.5) mm, rotated rx -180 ry 0 rz 90 deg; joints [8.565, -49.942, 87.644, 193.834, 38.521, -190.906]
  MoveL 558 to (-960, 200, 50) mm, rotated rx 180 ry 0 rz 90 deg; joints [8.565, -51.516, 87.353, 194.426, 36.712, -191.652]
  MoveL 559 to (-960, 250, 50) mm, rotated rx 180 ry 0 rz 90 deg; joints [8.782, -53.444, 90.717, 194.31, 38.147, -191.343]
  MoveL 560 to (-960, 250, -0.5) mm, rotated rx -180 ry 0 rz 90 deg; joints [8.782, -51.818, 91.009, 193.738, 40.007, -190.606]
  MoveL 561 to (-960, 250, 50) mm, rotated rx 180 ry 0 rz 90 deg; joints [8.782, -53.444, 90.717, 194.31, 38.147, -191.343]
  MoveL 562 to (-960, 300, 50) mm, rotated rx 180 ry 0 rz 90 deg; joints [9.01, -55.337, 93.986, 194.245, 39.525, -191.08]
  MoveL 563 to (-960, 300, -0.5) mm, rotated rx 180 ry 0 rz 90 deg; joints [9.01, -53.657, 94.279, 193.687, 41.44, -190.347]
  MoveL 564 to (-960, 300, 50) mm, rotated rx 180 ry 0 rz 90 deg; joints [9.01, -55.337, 93.986, 194.245, 39.525, -191.08]
  MoveL 565 to (-960, 350, 50) mm, rotated rx -180 ry 0 rz 90 deg; joints [9.25, -57.202, 97.171, 194.227, 40.85, -190.857]
  MoveL 566 to (-960, 350, -0.5) mm, rotated rx 180 ry 0 rz 90 deg; joints [9.25, -55.465, 97.466, 193.679, 42.822, -190.122]
  MoveL 567 to (-960, 350, 50) mm, rotated rx -180 ry 0 rz 90 deg; joints [9.25, -57.202, 97.171, 194.227, 40.85, -190.857]
  MoveL 568 to (-960, 400, 50) mm, rotated rx 180 ry 0 rz 90 deg; joints [9.504, -59.044, 100.278, 194.251, 42.123, -190.668]
  MoveL 569 to (-960, 400, -0.5) mm, rotated rx 180 ry 0 rz 90 deg; joints [9.504, -57.247, 100.577, 193.711, 44.157, -189.928]
  MoveL 570 to (-960, 400, 50) mm, rotated rx 180 ry 0 rz 90 deg; joints [9.504, -59.044, 100.278, 194.251, 42.123, -190.668]
  MoveL 571 to (-960, 450, 50) mm, rotated rx -180 ry 0 rz 90 deg; joints [9.771, -60.869, 103.316, 194.315, 43.348, -190.512]
  MoveL 572 to (-960, 450, -0.5) mm, rotated rx 180 ry 0 rz 90 deg; joints [9.771, -59.008, 103.618, 193.778, 45.447, -189.762]
  MoveL 573 to (-960, 450, 50) mm, rotated rx -180 ry 0 rz 90 deg; joints [9.771, -60.869, 103.316, 194.315, 43.348, -190.512]
  MoveL 574 to (-960, 500, 50) mm, rotated rx 180 ry 0 rz 90 deg; joints [10.054, -62.682, 106.289, 194.417, 44.524, -190.386]
  MoveL 575 to (-960, 500, -0.5) mm, rotated rx 180 ry 0 rz 90 deg; joints [10.054, -60.753, 106.597, 193.882, 46.692, -189.621]
  MoveL 576 to (-960, 500, 50) mm, rotated rx 180 ry 0 rz 90 deg; joints [10.054, -62.682, 106.289, 194.417, 44.524, -190.386]
  MoveL 577 to (-960, 550, 50) mm, rotated rx 180 ry 0 rz 90 deg; joints [10.354, -64.487, 109.204, 194.556, 45.652, -190.288]
  MoveL 578 to (-960, 550, -0.5) mm, rotated rx 180 ry 0 rz 90 deg; joints [10.354, -62.485, 109.517, 194.019, 47.895, -189.504]
  MoveL 579 to (-960, 550, 50) mm, rotated rx 180 ry 0 rz 90 deg; joints [10.354, -64.487, 109.204, 194.556, 45.652, -190.288]
  MoveL 580 to (-960, 600, 50) mm, rotated rx -180 ry 0 rz 90 deg; joints [10.672, -66.29, 112.065, 194.733, 46.732, -190.217]
  MoveL 581 to (-960, 600, -0.5) mm, rotated rx -180 ry 0 rz 90 deg; joints [10.672, -64.21, 112.384, 194.192, 49.055, -189.41]
  MoveL 582 to (-960, 600, 50) mm, rotated rx -180 ry 0 rz 90 deg; joints [10.672, -66.29, 112.065, 194.733, 46.732, -190.217]
  MoveL 583 to (-960, 650, 50) mm, rotated rx -180 ry 0 rz 90 deg; joints [11.01, -68.094, 114.875, 194.948, 47.764, -190.174]
  MoveL 584 to (-960, 650, -0.5) mm, rotated rx -180 ry 0 rz 90 deg; joints [11.01, -65.931, 115.202, 194.399, 50.173, -189.338]
  MoveL 585 to (-960, 650, 50) mm, rotated rx -180 ry 0 rz 90 deg; joints [11.01, -68.094, 114.875, 194.948, 47.764, -190.174]
  MoveL 586 to (-960, 700, 50) mm, rotated rx -180 ry 0 rz 90 deg; joints [11.369, -69.906, 117.639, 195.201, 48.747, -190.158]
  MoveL 587 to (-960, 700, -0.5) mm, rotated rx -180 ry 0 rz 90 deg; joints [11.369, -67.654, 117.975, 194.642, 51.248, -189.288]
  MoveL 588 to (-960, 700, 50) mm, rotated rx -180 ry 0 rz 90 deg; joints [11.369, -69.906, 117.639, 195.201, 48.747, -190.158]
  MoveL 589 to (-960, 750, 50) mm, rotated rx -180 ry 0 rz 90 deg; joints [11.752, -71.73, 120.359, 195.495, 49.678, -190.17]
  MoveL 590 to (-960, 750, -0.5) mm, rotated rx -180 ry 0 rz 90 deg; joints [11.752, -69.381, 120.704, 194.922, 52.278, -189.26]
  MoveL 591 to (-960, 750, 50) mm, rotated rx -180 ry 0 rz 90 deg; joints [11.752, -71.73, 120.359, 195.495, 49.678, -190.17]
  MoveL 592 to (-960, 800, 50) mm, rotated rx -180 ry 0 rz 90 deg; joints [12.162, -73.572, 123.037, 195.832, 50.556, -190.213]
  MoveL 593 to (-960, 800, -0.5) mm, rotated rx -180 ry 0 rz 90 deg; joints [12.162, -71.12, 123.394, 195.242, 53.263, -189.257]
  MoveL 594 to (-960, 800, 50) mm, rotated rx -180 ry 0 rz 90 deg; joints [12.162, -73.572, 123.037, 195.832, 50.556, -190.213]
  MoveL 595 to (-960, 850, 50) mm, rotated rx 180 ry 0 rz 90 deg; joints [12.601, -75.44, 125.677, 196.215, 51.376, -190.289]
  MoveL 596 to (-960, 850, -0.5) mm, rotated rx 180 ry 0 rz 90 deg; joints [12.601, -72.874, 126.046, 195.604, 54.199, -189.278]
  MoveL 597 to (-960, 850, 50) mm, rotated rx 180 ry 0 rz 90 deg; joints [12.601, -75.44, 125.677, 196.215, 51.376, -190.289]
  MoveL 598 to (-960, 900, 50) mm, rotated rx 180 ry 0 rz 90 deg; joints [13.072, -77.339, 128.28, 196.648, 52.136, -190.4]
  MoveL 599 to (-960, 900, -0.5) mm, rotated rx 180 ry 0 rz 90 deg; joints [13.072, -74.65, 128.663, 196.012, 55.084, -189.328]
  MoveL 600 to (-960, 900, 50) mm, rotated rx 180 ry 0 rz 90 deg; joints [13.072, -77.339, 128.28, 196.648, 52.136, -190.4]
  MoveL 601 to (-960, 950, 50) mm, rotated rx -180 ry 0 rz 90 deg; joints [13.579, -79.278, 130.847, 197.137, 52.83, -190.553]
  MoveL 602 to (-960, 950, -0.5) mm, rotated rx 180 ry 0 rz 90 deg; joints [13.579, -76.454, 131.246, 196.469, 55.914, -189.407]
  MoveL 603 to (-960, 950, 50) mm, rotated rx -180 ry 0 rz 90 deg; joints [13.579, -79.278, 130.847, 197.137, 52.83, -190.553]
  MoveL 604 to (-960, 1000, 50) mm, rotated rx 180 ry 0 rz 90 deg; joints [14.127, -81.266, 133.38, 197.687, 53.451, -190.753]
  MoveL 605 to (-960, 1000, -0.5) mm, rotated rx 180 ry 0 rz 90 deg; joints [14.127, -78.295, 133.797, 196.982, 56.684, -189.522]
  MoveL 606 to (-960, 1000, 50) mm, rotated rx 180 ry 0 rz 90 deg; joints [14.127, -81.266, 133.38, 197.687, 53.451, -190.753]
  MoveL 607 to (-960, 1050, 50) mm, rotated rx -180 ry 0 rz 90 deg; joints [14.719, -83.315, 135.88, 198.306, 53.991, -191.007]
  MoveL 608 to (-960, 1050, -0.5) mm, rotated rx -180 ry 0 rz 90 deg; joints [14.719, -80.182, 136.316, 197.556, 57.387, -189.677]
  MoveL 609 to (-960, 1050, 50) mm, rotated rx -180 ry 0 rz 90 deg; joints [14.719, -83.315, 135.88, 198.306, 53.991, -191.007]
  MoveL 610 to (-960, 1100, 50) mm, rotated rx 180 ry 0 rz 90 deg; joints [15.362, -85.437, 138.347, 199.004, 54.442, -191.325]
  MoveL 611 to (-960, 1100, -0.5) mm, rotated rx -180 ry 0 rz 90 deg; joints [15.362, -82.126, 138.806, 198.199, 58.015, -189.879]
  MoveL 612 to (-960, 1100, 50) mm, rotated rx 180 ry 0 rz 90 deg; joints [15.362, -85.437, 138.347, 199.004, 54.442, -191.325]
  MoveL 613 to (-960, 1150, 50) mm, rotated rx -180 ry 0 rz 90 deg; joints [16.062, -87.649, 140.782, 199.792, 54.792, -191.722]
  MoveL 614 to (-960, 1150, -0.5) mm, rotated rx -180 ry 0 rz 90 deg; joints [16.062, -84.14, 141.266, 198.922, 58.56, -190.138]
  MoveL 615 to (-960, 1150, 50) mm, rotated rx -180 ry 0 rz 90 deg; joints [16.062, -87.649, 140.782, 199.792, 54.792, -191.722]
  MoveL 616 to (-960, 1200, 50) mm, rotated rx -180 ry 0 rz 90 deg; joints [16.826, -89.97, 143.183, 200.687, 55.027, -192.213]
  MoveL 617 to (-960, 1200, -0.5) mm, rotated rx 180 ry 0 rz 90 deg; joints [16.826, -86.241, 143.697, 199.736, 59.008, -190.466]
  MoveL 618 to (-960, 1200, 50) mm, rotated rx -180 ry 0 rz 90 deg; joints [16.826, -89.97, 143.183, 200.687, 55.027, -192.213]
  MoveL 619 to (-1030, 50, 50) mm, rotated rx -180 ry 0 rz 90 deg; joints [9.8, -44.991, 75.733, 198.671, 32.12, -195.971]
  MoveL 620 to (-1030, 50, -0.5) mm, rotated rx 180 ry 0 rz 90 deg; joints [9.8, -43.568, 76.031, 197.839, 33.754, -194.98]
  MoveL 621 to (-1030, 50, 50) mm, rotated rx -180 ry 0 rz 90 deg; joints [9.8, -44.991, 75.733, 198.671, 32.12, -195.971]
  MoveL 622 to (-1030, 100, 50) mm, rotated rx 180 ry 0 rz 90 deg; joints [10.03, -47.071, 79.472, 198.266, 33.756, -195.346]
  MoveL 623 to (-1030, 100, -0.5) mm, rotated rx 180 ry 0 rz 90 deg; joints [10.03, -45.603, 79.767, 197.482, 35.433, -194.393]
  MoveL 624 to (-1030, 100, 50) mm, rotated rx 180 ry 0 rz 90 deg; joints [10.03, -47.071, 79.472, 198.266, 33.756, -195.346]
  MoveL 625 to (-1030, 150, 50) mm, rotated rx 180 ry 0 rz 90 deg; joints [10.27, -49.09, 83.071, 197.962, 35.32, -194.816]
  MoveL 626 to (-1030, 150, -0.5) mm, rotated rx -180 ry 0 rz 90 deg; joints [10.27, -47.576, 83.364, 197.216, 37.042, -193.892]
  MoveL 627 to (-1030, 150, 50) mm, rotated rx 180 ry 0 rz 90 deg; joints [10.27, -49.09, 83.071, 197.962, 35.32, -194.816]
  MoveL 628 to (-1030, 200, 50) mm, rotated rx 180 ry 0 rz 90 deg; joints [10.522, -51.058, 86.548, 197.741, 36.82, -194.366]
  MoveL 629 to (-1030, 200, -0.5) mm, rotated rx 180 ry 0 rz 90 deg; joints [10.522, -49.496, 86.84, 197.025, 38.589, -193.46]
  MoveL 630 to (-1030, 200, 50) mm, rotated rx 180 ry 0 rz 90 deg; joints [10.522, -51.058, 86.548, 197.741, 36.82, -194.366]
  MoveL 631 to (-1030, 250, 50) mm, rotated rx -180 ry 0 rz 90 deg; joints [10.787, -52.983, 89.916, 197.593, 38.259, -193.981]
  MoveL 632 to (-1030, 250, -0.5) mm, rotated rx -180 ry 0 rz 90 deg; joints [10.787, -51.37, 90.208, 196.899, 40.078, -193.087]
  MoveL 633 to (-1030, 250, 50) mm, rotated rx -180 ry 0 rz 90 deg; joints [10.787, -52.983, 89.916, 197.593, 38.259, -193.981]
  MoveL 634 to (-1030, 300, 50) mm, rotated rx 180 ry 0 rz 90 deg; joints [11.065, -54.872, 93.187, 197.507, 39.643, -193.652]
  MoveL 635 to (-1030, 300, -0.5) mm, rotated rx 180 ry 0 rz 90 deg; joints [11.065, -53.206, 93.479, 196.832, 41.515, -192.763]
  MoveL 636 to (-1030, 300, 50) mm, rotated rx 180 ry 0 rz 90 deg; joints [11.065, -54.872, 93.187, 197.507, 39.643, -193.652]
  MoveL 637 to (-1030, 350, 50) mm, rotated rx 180 ry 0 rz 90 deg; joints [11.358, -56.731, 96.37, 197.477, 40.975, -193.372]
  MoveL 638 to (-1030, 350, -0.5) mm, rotated rx -180 ry 0 rz 90 deg; joints [11.358, -55.009, 96.665, 196.815, 42.902, -192.483]
  MoveL 639 to (-1030, 350, 50) mm, rotated rx 180 ry 0 rz 90 deg; joints [11.358, -56.731, 96.37, 197.477, 40.975, -193.372]
  MoveL 640 to (-1030, 400, 50) mm, rotated rx -180 ry 0 rz 90 deg; joints [11.666, -58.565, 99.475, 197.5, 42.257, -193.135]
  MoveL 641 to (-1030, 400, -0.5) mm, rotated rx 180 ry 0 rz 90 deg; joints [11.666, -56.784, 99.772, 196.847, 44.243, -192.24]
  MoveL 642 to (-1030, 400, 50) mm, rotated rx -180 ry 0 rz 90 deg; joints [11.666, -58.565, 99.475, 197.5, 42.257, -193.135]
  MoveL 643 to (-1030, 450, 50) mm, rotated rx -180 ry 0 rz 90 deg; joints [11.991, -60.381, 102.508, 197.57, 43.491, -192.938]
  MoveL 644 to (-1030, 450, -0.5) mm, rotated rx 180 ry 0 rz 90 deg; joints [11.991, -58.537, 102.809, 196.924, 45.54, -192.031]
  MoveL 645 to (-1030, 450, 50) mm, rotated rx -180 ry 0 rz 90 deg; joints [11.991, -60.381, 102.508, 197.57, 43.491, -192.938]
  MoveL 646 to (-1030, 500, 50) mm, rotated rx 180 ry 0 rz 90 deg; joints [12.335, -62.182, 105.475, 197.688, 44.678, -192.776]
  MoveL 647 to (-1030, 500, -0.5) mm, rotated rx -180 ry 0 rz 90 deg; joints [12.335, -60.272, 105.78, 197.043, 46.793, -191.853]
  MoveL 648 to (-1030, 500, 50) mm, rotated rx 180 ry 0 rz 90 deg; joints [12.335, -62.182, 105.475, 197.688, 44.678, -192.776]
  MoveL 649 to (-1030, 550, 50) mm, rotated rx 180 ry 0 rz 90 deg; joints [12.699, -63.974, 108.381, 197.85, 45.82, -192.649]
  MoveL 650 to (-1030, 550, -0.5) mm, rotated rx -180 ry 0 rz 90 deg; joints [12.699, -61.993, 108.692, 197.204, 48.006, -191.704]
  MoveL 651 to (-1030, 550, 50) mm, rotated rx 180 ry 0 rz 90 deg; joints [12.699, -63.974, 108.381, 197.85, 45.82, -192.649]
  MoveL 652 to (-1030, 600, 50) mm, rotated rx -180 ry 0 rz 90 deg; joints [13.084, -65.761, 111.231, 198.057, 46.916, -192.554]
  MoveL 653 to (-1030, 600, -0.5) mm, rotated rx 180 ry 0 rz 90 deg; joints [13.084, -63.705, 111.549, 197.407, 49.177, -191.582]
  MoveL 654 to (-1030, 600, 50) mm, rotated rx -180 ry 0 rz 90 deg; joints [13.084, -65.761, 111.231, 198.057, 46.916, -192.554]
  MoveL 655 to (-1030, 650, 50) mm, rotated rx 180 ry 0 rz 90 deg; joints [13.493, -67.547, 114.03, 198.309, 47.966, -192.492]
  MoveL 656 to (-1030, 650, -0.5) mm, rotated rx -180 ry 0 rz 90 deg; joints [13.493, -65.411, 114.355, 197.651, 50.307, -191.488]
  MoveL 657 to (-1030, 650, 50) mm, rotated rx 180 ry 0 rz 90 deg; joints [13.493, -67.547, 114.03, 198.309, 47.966, -192.492]
  MoveL 658 to (-1030, 700, 50) mm, rotated rx 180 ry 0 rz 90 deg; joints [13.928, -69.338, 116.779, 198.607, 48.969, -192.463]
  MoveL 659 to (-1030, 700, -0.5) mm, rotated rx 180 ry 0 rz 90 deg; joints [13.928, -67.115, 117.113, 197.939, 51.397, -191.419]
  MoveL 660 to (-1030, 700, 50) mm, rotated rx 180 ry 0 rz 90 deg; joints [13.928, -69.338, 116.779, 198.607, 48.969, -192.463]
  MoveL 661 to (-1030, 750, 50) mm, rotated rx 180 ry 0 rz 90 deg; joints [14.391, -71.138, 119.484, 198.953, 49.925, -192.467]
  MoveL 662 to (-1030, 750, -0.5) mm, rotated rx -180 ry 0 rz 90 deg; joints [14.391, -68.822, 119.826, 198.271, 52.445, -191.378]
  MoveL 663 to (-1030, 750, 50) mm, rotated rx 180 ry 0 rz 90 deg; joints [14.391, -71.138, 119.484, 198.953, 49.925, -192.467]
  MoveL 664 to (-1030, 800, 50) mm, rotated rx -180 ry 0 rz 90 deg; joints [14.885, -72.953, 122.145, 199.35, 50.832, -192.506]
  MoveL 665 to (-1030, 800, -0.5) mm, rotated rx 180 ry 0 rz 90 deg; joints [14.885, -70.536, 122.497, 198.649, 53.451, -191.364]
  MoveL 666 to (-1030, 800, 50) mm, rotated rx -180 ry 0 rz 90 deg; joints [14.885, -72.953, 122.145, 199.35, 50.832, -192.506]
  MoveL 667 to (-1030, 850, 50) mm, rotated rx -180 ry 0 rz 90 deg; joints [15.414, -74.788, 124.765, 199.801, 51.686, -192.583]
  MoveL 668 to (-1030, 850, -0.5) mm, rotated rx 180 ry 0 rz 90 deg; joints [15.414, -72.263, 125.129, 199.077, 54.412, -191.379]
  MoveL 669 to (-1030, 850, 50) mm, rotated rx -180 ry 0 rz 90 deg; joints [15.414, -74.788, 124.765, 199.801, 51.686, -192.583]
  MoveL 670 to (-1030, 900, 50) mm, rotated rx 180 ry 0 rz 90 deg; joints [15.981, -76.65, 127.346, 200.309, 52.486, -192.701]
  MoveL 671 to (-1030, 900, -0.5) mm, rotated rx 180 ry 0 rz 90 deg; joints [15.981, -74.007, 127.724, 199.558, 55.326, -191.426]
  MoveL 672 to (-1030, 900, 50) mm, rotated rx 180 ry 0 rz 90 deg; joints [15.981, -76.65, 127.346, 200.309, 52.486, -192.701]
  MoveL 673 to (-1030, 950, 50) mm, rotated rx 180 ry 0 rz 90 deg; joints [16.589, -78.546, 129.889, 200.881, 53.227, -192.865]
  MoveL 674 to (-1030, 950, -0.5) mm, rotated rx -180 ry 0 rz 90 deg; joints [16.589, -75.774, 130.282, 200.097, 56.191, -191.508]
  MoveL 675 to (-1030, 950, 50) mm, rotated rx 180 ry 0 rz 90 deg; joints [16.589, -78.546, 129.889, 200.881, 53.227, -192.865]
  MoveL 676 to (-1030, 1000, 50) mm, rotated rx -180 ry 0 rz 90 deg; joints [17.244, -80.483, 132.396, 201.523, 53.904, -193.08]
  MoveL 677 to (-1030, 1000, -0.5) mm, rotated rx -180 ry 0 rz 90 deg; joints [17.244, -77.572, 132.805, 200.7, 57.002, -191.628]
  MoveL 678 to (-1030, 1000, 50) mm, rotated rx -180 ry 0 rz 90 deg; joints [17.244, -80.483, 132.396, 201.523, 53.904, -193.08]
  MoveL 679 to (-1030, 1050, 50) mm, rotated rx 180 ry 0 rz 90 deg; joints [17.952, -82.473, 134.867, 202.243, 54.513, -193.355]
  MoveL 680 to (-1030, 1050, -0.5) mm, rotated rx 180 ry 0 rz 90 deg; joints [17.952, -79.408, 135.294, 201.372, 57.756, -191.793]
  MoveL 681 to (-1030, 1050, 50) mm, rotated rx 180 ry 0 rz 90 deg; joints [17.952, -82.473, 134.867, 202.243, 54.513, -193.355]
  MoveL 682 to (-1030, 1100, 50) mm, rotated rx 180 ry 0 rz 90 deg; joints [18.718, -84.524, 137.302, 203.05, 55.046, -193.7]
  MoveL 683 to (-1030, 1100, -0.5) mm, rotated rx -180 ry 0 rz 90 deg; joints [18.718, -81.292, 137.751, 202.123, 58.445, -192.01]
  MoveL 684 to (-1030, 1100, 50) mm, rotated rx 180 ry 0 rz 90 deg; joints [18.718, -84.524, 137.302, 203.05, 55.046, -193.7]
  MoveL 685 to (-1030, 1150, 50) mm, rotated rx -180 ry 0 rz 90 deg; joints [19.549, -86.652, 139.702, 203.957, 55.496, -194.128]
  MoveL 686 to (-1030, 1150, -0.5) mm, rotated rx -180 ry 0 rz 90 deg; joints [19.549, -83.234, 140.174, 202.961, 59.065, -192.287]
  MoveL 687 to (-1030, 1150, 50) mm, rotated rx -180 ry 0 rz 90 deg; joints [19.549, -86.652, 139.702, 203.957, 55.496, -194.128]
  MoveL 688 to (-1030, 1200, 50) mm, rotated rx 180 ry 0 rz 90 deg; joints [20.455, -88.87, 142.065, 204.978, 55.853, -194.654]
  MoveL 689 to (-1030, 1200, -0.5) mm, rotated rx -180 ry 0 rz 90 deg; joints [20.455, -85.248, 142.565, 203.9, 59.606, -192.637]
  MoveL 690 to (-1030, 1200, 50) mm, rotated rx 180 ry 0 rz 90 deg; joints [20.455, -88.87, 142.065, 204.978, 55.853, -194.654]
  MoveL 691 to (-1100, 50, 50) mm, rotated rx 180 ry 0 rz 90 deg; joints [11.608, -44.43, 74.72, 202.16, 32.239, -199.008]
  MoveL 692 to (-1100, 50, -0.5) mm, rotated rx 180 ry 0 rz 90 deg; joints [11.608, -43.019, 75.019, 201.188, 33.829, -197.849]
  MoveL 693 to (-1100, 50, 50) mm, rotated rx 180 ry 0 rz 90 deg; joints [11.608, -44.43, 74.72, 202.16, 32.239, -199.008]
  MoveL 694 to (-1100, 100, 50) mm, rotated rx 180 ry 0 rz 90 deg; joints [11.878, -46.515, 78.476, 201.67, 33.876, -198.257]
  MoveL 695 to (-1100, 100, -0.5) mm, rotated rx 180 ry 0 rz 90 deg; joints [11.878, -45.06, 78.772, 200.754, 35.509, -197.144]
  MoveL 696 to (-1100, 100, 50) mm, rotated rx 180 ry 0 rz 90 deg; joints [11.878, -46.515, 78.476, 201.67, 33.876, -198.257]
  MoveL 697 to (-1100, 150, 50) mm, rotated rx 180 ry 0 rz 90 deg; joints [12.16, -48.537, 82.088, 201.299, 35.443, -197.621]
  MoveL 698 to (-1100, 150, -0.5) mm, rotated rx -180 ry 0 rz 90 deg; joints [12.16, -47.036, 82.381, 200.429, 37.12, -196.541]
  MoveL 699 to (-1100, 150, 50) mm, rotated rx 180 ry 0 rz 90 deg; joints [12.16, -48.537, 82.088, 201.299, 35.443, -197.621]
  MoveL 700 to (-1100, 200, 50) mm, rotated rx -180 ry 0 rz 90 deg; joints [12.456, -50.505, 85.573, 201.029, 36.946, -197.079]
  MoveL 701 to (-1100, 200, -0.5) mm, rotated rx 180 ry 0 rz 90 deg; joints [12.456, -48.956, 85.865, 200.194, 38.669, -196.022]
  MoveL 702 to (-1100, 200, 50) mm, rotated rx -180 ry 0 rz 90 deg; joints [12.456, -50.505, 85.573, 201.029, 36.946, -197.079]
  MoveL 703 to (-1100, 250, 50) mm, rotated rx -180 ry 0 rz 90 deg; joints [12.766, -52.427, 88.947, 200.843, 38.391, -196.616]
  MoveL 704 to (-1100, 250, -0.5) mm, rotated rx 180 ry 0 rz 90 deg; joints [12.766, -50.829, 89.238, 200.036, 40.162, -195.573]
  MoveL 705 to (-1100, 250, 50) mm, rotated rx -180 ry 0 rz 90 deg; joints [12.766, -52.427, 88.947, 200.843, 38.391, -196.616]
  MoveL 706 to (-1100, 300, 50) mm, rotated rx -180 ry 0 rz 90 deg; joints [13.092, -54.311, 92.22, 200.732, 39.782, -196.219]
  MoveL 707 to (-1100, 300, -0.5) mm, rotated rx 180 ry 0 rz 90 deg; joints [13.092, -52.661, 92.512, 199.947, 41.603, -195.183]
  MoveL 708 to (-1100, 300, 50) mm, rotated rx -180 ry 0 rz 90 deg; joints [13.092, -54.311, 92.22, 200.732, 39.782, -196.219]
  MoveL 709 to (-1100, 350, 50) mm, rotated rx 180 ry 0 rz 90 deg; joints [13.435, -56.164, 95.403, 200.688, 41.121, -195.88]
  MoveL 710 to (-1100, 350, -0.5) mm, rotated rx 180 ry 0 rz 90 deg; joints [13.435, -54.459, 95.697, 199.919, 42.996, -194.844]
  MoveL 711 to (-1100, 350, 50) mm, rotated rx 180 ry 0 rz 90 deg; joints [13.435, -56.164, 95.403, 200.688, 41.121, -195.88]
  MoveL 712 to (-1100, 400, 50) mm, rotated rx 180 ry 0 rz 90 deg; joints [13.795, -57.99, 98.505, 200.704, 42.413, -195.591]
  MoveL 713 to (-1100, 400, -0.5) mm, rotated rx 180 ry 0 rz 90 deg; joints [13.795, -56.228, 98.802, 199.947, 44.343, -194.55]
  MoveL 714 to (-1100, 400, 50) mm, rotated rx 180 ry 0 rz 90 deg; joints [13.795, -57.99, 98.505, 200.704, 42.413, -195.591]
  MoveL 715 to (-1100, 450, 50) mm, rotated rx 180 ry 0 rz 90 deg; joints [14.175, -59.795, 101.533, 200.777, 43.658, -195.349]
  MoveL 716 to (-1100, 450, -0.5) mm, rotated rx -180 ry 0 rz 90 deg; joints [14.175, -57.972, 101.833, 200.028, 45.648, -194.296]
  MoveL 717 to (-1100, 450, 50) mm, rotated rx 180 ry 0 rz 90 deg; joints [14.175, -59.795, 101.533, 200.777, 43.658, -195.349]
  MoveL 718 to (-1100, 500, 50) mm, rotated rx 180 ry 0 rz 90 deg; joints [14.577, -61.583, 104.492, 200.904, 44.858, -195.15]
  MoveL 719 to (-1100, 500, -0.5) mm, rotated rx -180 ry 0 rz 90 deg; joints [14.577, -59.696, 104.796, 200.159, 46.91, -194.079]
  MoveL 720 to (-1100, 500, 50) mm, rotated rx 180 ry 0 rz 90 deg; joints [14.577, -61.583, 104.492, 200.904, 44.858, -195.15]
  MoveL 721 to (-1100, 550, 50) mm, rotated rx 180 ry 0 rz 90 deg; joints [15.001, -63.36, 107.389, 201.084, 46.014, -194.99]
  MoveL 722 to (-1100, 550, -0.5) mm, rotated rx -180 ry 0 rz 90 deg; joints [15.001, -61.404, 107.698, 200.339, 48.133, -193.896]
  MoveL 723 to (-1100, 550, 50) mm, rotated rx 180 ry 0 rz 90 deg; joints [15.001, -63.36, 107.389, 201.084, 46.014, -194.99]
  MoveL 724 to (-1100, 600, 50) mm, rotated rx -180 ry 0 rz 90 deg; joints [15.45, -65.128, 110.228, 201.315, 47.127, -194.867]
  MoveL 725 to (-1100, 600, -0.5) mm, rotated rx 180 ry 0 rz 90 deg; joints [15.45, -63.1, 110.543, 200.566, 49.317, -193.744]
  MoveL 726 to (-1100, 600, 50) mm, rotated rx -180 ry 0 rz 90 deg; joints [15.45, -65.128, 110.228, 201.315, 47.127, -194.867]
  MoveL 727 to (-1100, 650, 50) mm, rotated rx -180 ry 0 rz 90 deg; joints [15.926, -66.894, 113.013, 201.598, 48.198, -194.782]
  MoveL 728 to (-1100, 650, -0.5) mm, rotated rx -180 ry 0 rz 90 deg; joints [15.926, -64.787, 113.335, 200.842, 50.462, -193.623]
  MoveL 729 to (-1100, 650, 50) mm, rotated rx -180 ry 0 rz 90 deg; joints [15.926, -66.894, 113.013, 201.598, 48.198, -194.782]
  MoveL 730 to (-1100, 700, 50) mm, rotated rx 180 ry 0 rz 90 deg; joints [16.431, -68.661, 115.747, 201.933, 49.224, -194.734]
  MoveL 731 to (-1100, 700, -0.5) mm, rotated rx -180 ry 0 rz 90 deg; joints [16.431, -66.471, 116.076, 201.167, 51.568, -193.533]
  MoveL 732 to (-1100, 700, 50) mm, rotated rx 180 ry 0 rz 90 deg; joints [16.431, -68.661, 115.747, 201.933, 49.224, -194.734]
  MoveL 733 to (-1100, 750, 50) mm, rotated rx -180 ry 0 rz 90 deg; joints [16.969, -70.434, 118.433, 202.323, 50.207, -194.724]
  MoveL 734 to (-1100, 750, -0.5) mm, rotated rx 180 ry 0 rz 90 deg; joints [16.969, -68.154, 118.771, 201.543, 52.636, -193.473]
  MoveL 735 to (-1100, 750, 50) mm, rotated rx -180 ry 0 rz 90 deg; joints [16.969, -70.434, 118.433, 202.323, 50.207, -194.724]
  MoveL 736 to (-1100, 800, 50) mm, rotated rx -180 ry 0 rz 90 deg; joints [17.541, -72.217, 121.074, 202.77, 51.145, -194.753]
  MoveL 737 to (-1100, 800, -0.5) mm, rotated rx -180 ry 0 rz 90 deg; joints [17.541, -69.842, 121.422, 201.971, 53.664, -193.444]
  MoveL 738 to (-1100, 800, 50) mm, rotated rx -180 ry 0 rz 90 deg; joints [17.541, -72.217, 121.074, 202.77, 51.145, -194.753]
  MoveL 739 to (-1100, 850, 50) mm, rotated rx -180 ry 0 rz 90 deg; joints [18.153, -74.016, 123.671, 203.277, 52.036, -194.823]
  MoveL 740 to (-1100, 850, -0.5) mm, rotated rx -180 ry 0 rz 90 deg; joints [18.153, -71.537, 124.031, 202.456, 54.652, -193.448]
  MoveL 741 to (-1100, 850, 50) mm, rotated rx -180 ry 0 rz 90 deg; joints [18.153, -74.016, 123.671, 203.277, 52.036, -194.823]
  MoveL 742 to (-1100, 900, 50) mm, rotated rx 180 ry 0 rz 90 deg; joints [18.807, -75.836, 126.227, 203.848, 52.879, -194.937]
  MoveL 743 to (-1100, 900, -0.5) mm, rotated rx -180 ry 0 rz 90 deg; joints [18.807, -73.245, 126.599, 202.999, 55.598, -193.486]
  MoveL 744 to (-1100, 900, 50) mm, rotated rx 180 ry 0 rz 90 deg; joints [18.807, -75.836, 126.227, 203.848, 52.879, -194.937]
  MoveL 745 to (-1100, 950, 50) mm, rotated rx -180 ry 0 rz 90 deg; joints [19.508, -77.683, 128.743, 204.488, 53.67, -195.101]
  MoveL 746 to (-1100, 950, -0.5) mm, rotated rx -180 ry 0 rz 90 deg; joints [19.508, -74.971, 129.129, 203.607, 56.499, -193.562]
  MoveL 747 to (-1100, 950, 50) mm, rotated rx -180 ry 0 rz 90 deg; joints [19.508, -77.683, 128.743, 204.488, 53.67, -195.101]
  MoveL 748 to (-1100, 1000, 50) mm, rotated rx -180 ry 0 rz 90 deg; joints [20.26, -79.565, 131.219, 205.204, 54.408, -195.319]
  MoveL 749 to (-1100, 1000, -0.5) mm, rotated rx -180 ry 0 rz 90 deg; joints [20.26, -76.721, 131.621, 204.284, 57.355, -193.679]
  MoveL 750 to (-1100, 1000, 50) mm, rotated rx -180 ry 0 rz 90 deg; joints [20.26, -79.565, 131.219, 205.204, 54.408, -195.319]
  MoveL 751 to (-1100, 1050, 50) mm, rotated rx -180 ry 0 rz 90 deg; joints [21.071, -81.488, 133.657, 206.004, 55.088, -195.599]
  MoveL 752 to (-1100, 1050, -0.5) mm, rotated rx -180 ry 0 rz 90 deg; joints [21.071, -78.501, 134.076, 205.037, 58.161, -193.842]
  MoveL 753 to (-1100, 1050, 50) mm, rotated rx -180 ry 0 rz 90 deg; joints [21.071, -81.488, 133.657, 206.004, 55.088, -195.599]
  MoveL 754 to (-1100, 1100, 50) mm, rotated rx -180 ry 0 rz 90 deg; joints [21.946, -83.463, 136.057, 206.896, 55.706, -195.95]
  MoveL 755 to (-1100, 1100, -0.5) mm, rotated rx 180 ry 0 rz 90 deg; joints [21.946, -80.319, 136.494, 205.874, 58.915, -194.059]
  MoveL 756 to (-1100, 1100, 50) mm, rotated rx -180 ry 0 rz 90 deg; joints [21.946, -83.463, 136.057, 206.896, 55.706, -195.95]
